LIN {X 0,Y 523.334,Z 556.737,A -85,B 0,C 180,E1 -4767.691,E2 -4767.691} C_VEL
LIN {X 0,Y 523.25,Z 558.343,A -85,B 0,C 180,E1 -4769.23,E2 -4769.23} C_VEL
LIN {X 0,Y 523.25,Z 558.561,A -85,B 0,C 180,E1 -4769.999,E2 -4769.999} C_VEL
LIN {X 0,Y 523.274,Z 557.739,A -85,B 0,C 180,E1 -4771.539,E2 -4771.539} C_VEL
LIN {X 0,Y 523.334,Z 556.746,A -85,B 0,C 180,E1 -4772.308,E2 -4772.308} C_VEL
LIN {X 0,Y 523.367,Z 555.35,A -85,B 0,C 180,E1 -4773.078,E2 -4773.078} C_VEL
LIN {X 0,Y 523.424,Z 552.412,A -85,B 0,C 180,E1 -4774.234,E2 -4774.234} C_VEL
LIN {X 0,Y 523.461,Z 548.433,A -85,B 0,C 180,E1 -4775.392,E2 -4775.392} C_VEL
LIN {X 0,Y 523.514,Z 543.212,A -85,B 0,C 180,E1 -4776.572,E2 -4776.572} C_VEL
LIN {X 0,Y 523.646,Z 536.864,A -85,B 0,C 180,E1 -4777.712,E2 -4777.712} C_VEL
LIN {X 0,Y 523.814,Z 528.822,A -85,B 0,C 180,E1 -4778.875,E2 -4778.875} C_VEL
LIN {X 0,Y 524.043,Z 520.628,A -85,B 0,C 180,E1 -4779.845,E2 -4779.845} C_VEL
LIN {X 0,Y 524.325,Z 510.638,A -85,B 0,C 180,E1 -4780.815,E2 -4780.815} C_VEL
LIN {X 0,Y 524.619,Z 499.337,A -85,B 0,C 180,E1 -4781.691,E2 -4781.691} C_VEL
LIN {X 0,Y 524.85,Z 488.306,A -85,B 0,C 180,E1 -4782.371,E2 -4782.371} C_VEL
LIN {X 0,Y 525.115,Z 476.061,A -85,B 0,C 180,E1 -4782.954,E2 -4782.954} C_VEL
LIN {X 0,Y 525.349,Z 463.204,A -85,B 0,C 180,E1 -4783.391,E2 -4783.391} C_VEL
LIN {X 0,Y 525.549,Z 449.567,A -85,B 0,C 180,E1 -4783.681,E2 -4783.681} C_VEL
LIN {X 0,Y 525.854,Z 356.039,A -85,B 0,C 180,E1 -4784.969,E2 -4784.969} C_VEL
LIN {X 0,Y 524.306,Z 345.568,A -85,B 0,C 180,E1 -4785.178,E2 -4785.178} C_VEL
LIN {X 0,Y 524.738,Z 323.602,A -85,B 0,C 180,E1 -4788.526,E2 -4788.526} C_VEL
LIN {X 0,Y 525.158,Z 305.117,A -85,B 0,C 180,E1 -4791.387,E2 -4791.387} C_VEL
LIN {X 0,Y 525.426,Z 293.296,A -85,B 0,C 180,E1 -4793.239,E2 -4793.239} C_VEL
LIN {X 0,Y 523.993,Z 285.215,A -85,B 0,C 180,E1 -4794.621,E2 -4794.621} C_VEL
LIN {X 0,Y 523.978,Z 285.218,A -85,B 0,C 180,E1 -4797.718,E2 -4797.718} C_VEL
LIN {X 0,Y 523.942,Z 285.215,A -85,B 0,C 180,E1 -4800.854,E2 -4800.854} C_VEL
LIN {X 0,Y 523.958,Z 285.216,A -85,B 0,C 180,E1 -4803.734,E2 -4803.734} C_VEL
LIN {X 0,Y 523.916,Z 285.225,A -85,B 0,C 180,E1 -4806.403,E2 -4806.403} C_VEL
LIN {X 0,Y 523.916,Z 285.218,A -85,B 0,C 180,E1 -4809.084,E2 -4809.084} C_VEL
LIN {X 0,Y 523.95,Z 285.219,A -85,B 0,C 180,E1 -4812.118,E2 -4812.118} C_VEL
LIN {X 0,Y 523.95,Z 285.214,A -85,B 0,C 180,E1 -4815.308,E2 -4815.308} C_VEL
LIN {X 0,Y 523.956,Z 285.221,A -85,B 0,C 180,E1 -4818.688,E2 -4818.688} C_VEL
LIN {X 0,Y 523.912,Z 285.219,A -85,B 0,C 180,E1 -4821.898,E2 -4821.898} C_VEL
LIN {X 0,Y 523.927,Z 285.223,A -85,B 0,C 180,E1 -4824.909,E2 -4824.909} C_VEL
LIN {X 0,Y 523.935,Z 285.215,A -85,B 0,C 180,E1 -4827.678,E2 -4827.678} C_VEL
LIN {X 0,Y 523.955,Z 285.219,A -85,B 0,C 180,E1 -4830.674,E2 -4830.674} C_VEL
LIN {X 0,Y 523.969,Z 285.212,A -85,B 0,C 180,E1 -4833.728,E2 -4833.728} C_VEL
LIN {X 0,Y 523.928,Z 285.217,A -85,B 0,C 180,E1 -4836.27,E2 -4836.27} C_VEL
LIN {X 0,Y 523.937,Z 285.219,A -85,B 0,C 180,E1 -4838.766,E2 -4838.766} C_VEL
LIN {X 0,Y 523.942,Z 285.224,A -85,B 0,C 180,E1 -4841.22,E2 -4841.22} C_VEL
LIN {X 0,Y 523.927,Z 285.22,A -85,B 0,C 180,E1 -4843.639,E2 -4843.639} C_VEL
LIN {X 0,Y 523.936,Z 285.216,A -85,B 0,C 180,E1 -4846.028,E2 -4846.028} C_VEL
LIN {X 0,Y 524.002,Z 285.207,A -85,B 0,C 180,E1 -4848.394,E2 -4848.394} C_VEL
LIN {X 0,Y 523.998,Z 285.217,A -85,B 0,C 180,E1 -4851.516,E2 -4851.516} C_VEL
LIN {X 0,Y 524.074,Z 285.198,A -85,B 0,C 180,E1 -4854.614,E2 -4854.614} C_VEL
LIN {X 0,Y 524.1,Z 285.204,A -85,B 0,C 180,E1 -4857.694,E2 -4857.694} C_VEL
LIN {X 0,Y 524.112,Z 285.193,A -85,B 0,C 180,E1 -4860.768,E2 -4860.768} C_VEL
LIN {X 0,Y 524.064,Z 285.2,A -85,B 0,C 180,E1 -4863.075,E2 -4863.075} C_VEL
LIN {X 0,Y 524.018,Z 285.21,A -85,B 0,C 180,E1 -4866.159,E2 -4866.159} C_VEL
LIN {X 0,Y 523.994,Z 285.21,A -85,B 0,C 180,E1 -4868.484,E2 -4868.484} C_VEL
LIN {X 0,Y 523.992,Z 285.214,A -85,B 0,C 180,E1 -4871.74,E2 -4871.74} C_VEL
LIN {X 0,Y 523.982,Z 285.209,A -85,B 0,C 180,E1 -4875.052,E2 -4875.052} C_VEL
LIN {X 0,Y 523.954,Z 285.22,A -85,B 0,C 180,E1 -4877.969,E2 -4877.969} C_VEL
LIN {X 0,Y 523.962,Z 285.219,A -85,B 0,C 180,E1 -4880.411,E2 -4880.411} C_VEL
LIN {X 0,Y 523.901,Z 285.221,A -85,B 0,C 180,E1 -4882.894,E2 -4882.894} C_VEL
LIN {X 0,Y 523.921,Z 285.217,A -85,B 0,C 180,E1 -4885.421,E2 -4885.421} C_VEL
LIN {X 0,Y 523.944,Z 285.218,A -85,B 0,C 180,E1 -4888.001,E2 -4888.001} C_VEL
LIN {X 0,Y 523.936,Z 285.219,A -85,B 0,C 180,E1 -4890.855,E2 -4890.855} C_VEL
LIN {X 0,Y 523.951,Z 285.214,A -85,B 0,C 180,E1 -4893.735,E2 -4893.735} C_VEL
LIN {X 0,Y 523.895,Z 285.226,A -85,B 0,C 180,E1 -4896.402,E2 -4896.402} C_VEL
LIN {X 0,Y 523.906,Z 285.223,A -85,B 0,C 180,E1 -4899.086,E2 -4899.086} C_VEL
LIN {X 0,Y 523.931,Z 285.217,A -85,B 0,C 180,E1 -4902.121,E2 -4902.121} C_VEL
LIN {X 0,Y 523.934,Z 285.219,A -85,B 0,C 180,E1 -4905.311,E2 -4905.311} C_VEL
LIN {X 0,Y 523.89,Z 285.228,A -85,B 0,C 180,E1 -4906.895,E2 -4906.895} C_VEL
LIN {X 0,Y 523.21,Z 285.308,A -85,B 0,C 180,E1 -4907.536,E2 -4907.536} C_VEL
LIN {X 0,Y 520.359,Z 285.665,A -85,B 0,C 180,E1 -4908.578,E2 -4908.578} C_VEL
LIN {X 0,Y 517.96,Z 285.963,A -85,B 0,C 180,E1 -4909.417,E2 -4909.417} C_VEL
LIN {X 0,Y 516.935,Z 286.088,A -85,B 0,C 180,E1 -4910.065,E2 -4910.065} C_VEL
LIN {X 0,Y 516.853,Z 286.098,A -85,B 0,C 180,E1 -4910.284,E2 -4910.284} C_VEL
LIN {X 0,Y 516.849,Z 286.105,A -85,B 0,C 180,E1 -4913.253,E2 -4913.253} C_VEL
LIN {X 0,Y 516.88,Z 286.094,A -85,B 0,C 180,E1 -4916.12,E2 -4916.12} C_VEL
LIN {X 0,Y 516.877,Z 286.099,A -85,B 0,C 180,E1 -4918.939,E2 -4918.939} C_VEL
LIN {X 0,Y 516.842,Z 286.104,A -85,B 0,C 180,E1 -4921.581,E2 -4921.581} C_VEL
LIN {X 0,Y 516.856,Z 286.097,A -85,B 0,C 180,E1 -4924.208,E2 -4924.208} C_VEL
LIN {X 0,Y 516.855,Z 286.098,A -85,B 0,C 180,E1 -4926.777,E2 -4926.777} C_VEL
LIN {X 0,Y 516.94,Z 286.093,A -85,B 0,C 180,E1 -4929.733,E2 -4929.733} C_VEL
LIN {X 0,Y 516.884,Z 286.094,A -85,B 0,C 180,E1 -4932.595,E2 -4932.595} C_VEL
LIN {X 0,Y 516.933,Z 286.089,A -85,B 0,C 180,E1 -4935.031,E2 -4935.031} C_VEL
LIN {X 0,Y 516.921,Z 286.092,A -85,B 0,C 180,E1 -4938.233,E2 -4938.233} C_VEL
LIN {X 0,Y 516.918,Z 286.095,A -85,B 0,C 180,E1 -4941.4,E2 -4941.4} C_VEL
LIN {X 0,Y 516.984,Z 286.217,A -85,B 0,C 180,E1 -4944.271,E2 -4944.271} C_VEL
LIN {X 0,Y 517.421,Z 290.644,A -85,B 0,C 180,E1 -4945.131,E2 -4945.131} C_VEL
LIN {X 0,Y 517.224,Z 305.053,A -85,B 0,C 180,E1 -4947.859,E2 -4947.859} C_VEL
LIN {X 0,Y 517.167,Z 309.42,A -85,B 0,C 180,E1 -4948.687,E2 -4948.687} C_VEL
LIN {X 0,Y 519.14,Z 320.603,A -85,B 0,C 180,E1 -4948.91,E2 -4948.91} C_VEL
LIN {X 0,Y 518.649,Z 416.692,A -85,B 0,C 180,E1 -4950.267,E2 -4950.267} C_VEL
LIN {X 0,Y 518.394,Z 429.69,A -85,B 0,C 180,E1 -4950.607,E2 -4950.607} C_VEL
LIN {X 0,Y 518.188,Z 442.692,A -85,B 0,C 180,E1 -4951.118,E2 -4951.118} C_VEL
LIN {X 0,Y 517.913,Z 454.471,A -85,B 0,C 180,E1 -4951.75,E2 -4951.75} C_VEL
LIN {X 0,Y 517.589,Z 465.783,A -85,B 0,C 180,E1 -4952.53,E2 -4952.53} C_VEL
LIN {X 0,Y 517.331,Z 475.987,A -85,B 0,C 180,E1 -4953.408,E2 -4953.408} C_VEL
LIN {X 0,Y 517.031,Z 484.379,A -85,B 0,C 180,E1 -4954.288,E2 -4954.288} C_VEL
LIN {X 0,Y 516.788,Z 493.475,A -85,B 0,C 180,E1 -4955.463,E2 -4955.463} C_VEL
LIN {X 0,Y 516.584,Z 501.205,A -85,B 0,C 180,E1 -4956.709,E2 -4956.709} C_VEL
LIN {X 0,Y 516.46,Z 506.722,A -85,B 0,C 180,E1 -4957.822,E2 -4957.822} C_VEL
LIN {X 0,Y 516.359,Z 511.397,A -85,B 0,C 180,E1 -4959.006,E2 -4959.006} C_VEL
LIN {X 0,Y 516.319,Z 514.967,A -85,B 0,C 180,E1 -4960.193,E2 -4960.193} C_VEL
LIN {X 0,Y 516.287,Z 517.639,A -85,B 0,C 180,E1 -4961.447,E2 -4961.447} C_VEL
LIN {X 0,Y 516.182,Z 519.129,A -85,B 0,C 180,E1 -4962.583,E2 -4962.583} C_VEL
LIN {X 0,Y 516.178,Z 519.7,A -85,B 0,C 180,E1 -4963.384,E2 -4963.384} C_VEL
LIN {X 0,Y 516.206,Z 519.621,A -85,B 0,C 180,E1 -4964.839,E2 -4964.839} C_VEL
LIN {X 0,Y 516.143,Z 518.833,A -85,B 0,C 180,E1 -4965.803,E2 -4965.803} C_VEL
LIN {X 0,Y 516.189,Z 517.703,A -85,B 0,C 180,E1 -4966.614,E2 -4966.614} C_VEL
LIN {X 0,Y 516.277,Z 515.579,A -85,B 0,C 180,E1 -4967.654,E2 -4967.654} C_VEL
LIN {X 0,Y 516.357,Z 511.48,A -85,B 0,C 180,E1 -4969.066,E2 -4969.066} C_VEL
LIN {X 0,Y 516.511,Z 506.399,A -85,B 0,C 180,E1 -4970.343,E2 -4970.343} C_VEL
LIN {X 0,Y 516.581,Z 500.268,A -85,B 0,C 180,E1 -4971.551,E2 -4971.551} C_VEL
LIN {X 0,Y 516.861,Z 492.303,A -85,B 0,C 180,E1 -4972.801,E2 -4972.801} C_VEL
LIN {X 0,Y 517.045,Z 483.958,A -85,B 0,C 180,E1 -4973.853,E2 -4973.853} C_VEL
LIN {X 0,Y 517.331,Z 473.616,A -85,B 0,C 180,E1 -4974.907,E2 -4974.907} C_VEL
LIN {X 0,Y 517.645,Z 463.336,A -85,B 0,C 180,E1 -4975.751,E2 -4975.751} C_VEL
LIN {X 0,Y 518.018,Z 451.513,A -85,B 0,C 180,E1 -4976.516,E2 -4976.516} C_VEL
LIN {X 0,Y 518.229,Z 439.172,A -85,B 0,C 180,E1 -4977.13,E2 -4977.13} C_VEL
LIN {X 0,Y 518.434,Z 426.616,A -85,B 0,C 180,E1 -4977.583,E2 -4977.583} C_VEL
LIN {X 0,Y 518.598,Z 413.993,A -85,B 0,C 180,E1 -4977.875,E2 -4977.875} C_VEL
LIN {X 0,Y 519.041,Z 319.422,A -85,B 0,C 180,E1 -4979.201,E2 -4979.201} C_VEL
LIN {X 0,Y 517.209,Z 309.191,A -85,B 0,C 180,E1 -4979.426,E2 -4979.426} C_VEL
LIN {X 0,Y 517.372,Z 293.368,A -85,B 0,C 180,E1 -4982.31,E2 -4982.31} C_VEL
LIN {X 0,Y 517.178,Z 287.47,A -85,B 0,C 180,E1 -4983.392,E2 -4983.392} C_VEL
LIN {X 0,Y 516.938,Z 286.096,A -85,B 0,C 180,E1 -4983.672,E2 -4983.672} C_VEL
LIN {X 0,Y 516.879,Z 286.098,A -85,B 0,C 180,E1 -4986.746,E2 -4986.746} C_VEL
LIN {X 0,Y 516.884,Z 286.096,A -85,B 0,C 180,E1 -4989.721,E2 -4989.721} C_VEL
LIN {X 0,Y 516.914,Z 286.093,A -85,B 0,C 180,E1 -4991.775,E2 -4991.775} C_VEL
LIN {X 0,Y 516.897,Z 286.097,A -85,B 0,C 180,E1 -4995.007,E2 -4995.007} C_VEL
LIN {X 0,Y 516.915,Z 286.098,A -85,B 0,C 180,E1 -4998.399,E2 -4998.399} C_VEL
LIN {X 0,Y 516.881,Z 286.096,A -85,B 0,C 180,E1 -5001.284,E2 -5001.284} C_VEL
LIN {X 0,Y 516.872,Z 286.098,A -85,B 0,C 180,E1 -5004.219,E2 -5004.219} C_VEL
LIN {X 0,Y 516.895,Z 286.1,A -85,B 0,C 180,E1 -5007.053,E2 -5007.053} C_VEL
LIN {X 0,Y 516.892,Z 286.092,A -85,B 0,C 180,E1 -5009.796,E2 -5009.796} C_VEL
LIN {X 0,Y 516.926,Z 286.09,A -85,B 0,C 180,E1 -5012.467,E2 -5012.467} C_VEL
LIN {X 0,Y 516.909,Z 286.099,A -85,B 0,C 180,E1 -5015.072,E2 -5015.072} C_VEL
LIN {X 0,Y 516.885,Z 286.094,A -85,B 0,C 180,E1 -5018.462,E2 -5018.462} C_VEL
LIN {X 0,Y 516.901,Z 286.094,A -85,B 0,C 180,E1 -5020.955,E2 -5020.955} C_VEL
LIN {X 0,Y 516.914,Z 286.099,A -85,B 0,C 180,E1 -5023.41,E2 -5023.41} C_VEL
LIN {X 0,Y 516.894,Z 286.096,A -85,B 0,C 180,E1 -5025.834,E2 -5025.834} C_VEL
LIN {X 0,Y 516.966,Z 286.085,A -85,B 0,C 180,E1 -5028.234,E2 -5028.234} C_VEL
LIN {X 0,Y 516.967,Z 286.085,A -85,B 0,C 180,E1 -5031.4,E2 -5031.4} C_VEL
LIN {X 0,Y 517.002,Z 286.088,A -85,B 0,C 180,E1 -5033.757,E2 -5033.757} C_VEL
LIN {X 0,Y 517.012,Z 286.076,A -85,B 0,C 180,E1 -5036.883,E2 -5036.883} C_VEL
LIN {X 0,Y 517.085,Z 286.074,A -85,B 0,C 180,E1 -5040,E2 -5040} C_VEL
LIN {X 0,Y 517.012,Z 286.077,A -85,B 0,C 180,E1 -5043.117,E2 -5043.117} C_VEL
LIN {X 0,Y 517.002,Z 286.084,A -85,B 0,C 180,E1 -5046.243,E2 -5046.243} C_VEL
LIN {X 0,Y 516.945,Z 286.086,A -85,B 0,C 180,E1 -5049.389,E2 -5049.389} C_VEL
LIN {X 0,Y 516.951,Z 286.083,A -85,B 0,C 180,E1 -5051.807,E2 -5051.807} C_VEL
LIN {X 0,Y 516.944,Z 286.085,A -85,B 0,C 180,E1 -5055.146,E2 -5055.146} C_VEL
LIN {X 0,Y 516.924,Z 286.093,A -85,B 0,C 180,E1 -5058.222,E2 -5058.222} C_VEL
LIN {X 0,Y 516.912,Z 286.096,A -85,B 0,C 180,E1 -5060.702,E2 -5060.702} C_VEL
LIN {X 0,Y 516.903,Z 286.093,A -85,B 0,C 180,E1 -5064.072,E2 -5064.072} C_VEL
LIN {X 0,Y 516.924,Z 286.093,A -85,B 0,C 180,E1 -5066.658,E2 -5066.658} C_VEL
LIN {X 0,Y 516.911,Z 286.089,A -85,B 0,C 180,E1 -5069.524,E2 -5069.524} C_VEL
LIN {X 0,Y 516.894,Z 286.096,A -85,B 0,C 180,E1 -5072.543,E2 -5072.543} C_VEL
LIN {X 0,Y 516.865,Z 286.102,A -85,B 0,C 180,E1 -5075.33,E2 -5075.33} C_VEL
LIN {X 0,Y 516.881,Z 286.095,A -85,B 0,C 180,E1 -5077.943,E2 -5077.943} C_VEL
LIN {X 0,Y 516.884,Z 286.096,A -85,B 0,C 180,E1 -5080.742,E2 -5080.742} C_VEL
LIN {X 0,Y 516.883,Z 286.097,A -85,B 0,C 180,E1 -5082.832,E2 -5082.832} C_VEL
LIN {X 0,Y 516.896,Z 286.097,A -85,B 0,C 180,E1 -5085.007,E2 -5085.007} C_VEL
LIN {X 0,Y 516.915,Z 286.091,A -85,B 0,C 180,E1 -5088.399,E2 -5088.399} C_VEL
LIN {X 0,Y 516.882,Z 286.097,A -85,B 0,C 180,E1 -5091.284,E2 -5091.284} C_VEL
LIN {X 0,Y 516.873,Z 286.098,A -85,B 0,C 180,E1 -5094.22,E2 -5094.22} C_VEL
LIN {X 0,Y 516.897,Z 286.092,A -85,B 0,C 180,E1 -5097.053,E2 -5097.053} C_VEL
LIN {X 0,Y 516.895,Z 286.101,A -85,B 0,C 180,E1 -5099.796,E2 -5099.796} C_VEL
LIN {X 0,Y 516.927,Z 286.095,A -85,B 0,C 180,E1 -5102.467,E2 -5102.467} C_VEL
LIN {X 0,Y 516.968,Z 286.253,A -85,B 0,C 180,E1 -5105.337,E2 -5105.337} C_VEL
LIN {X 0,Y 518.473,Z 295.27,A -85,B 0,C 180,E1 -5106.852,E2 -5106.852} C_VEL
LIN {X 0,Y 517.947,Z 315.172,A -85,B 0,C 180,E1 -5109.977,E2 -5109.977} C_VEL
LIN {X 0,Y 517.471,Z 333.541,A -85,B 0,C 180,E1 -5112.818,E2 -5112.818} C_VEL
LIN {X 0,Y 517.285,Z 345.531,A -85,B 0,C 180,E1 -5114.635,E2 -5114.635} C_VEL
LIN {X 0,Y 519.028,Z 357.668,A -85,B 0,C 180,E1 -5114.857,E2 -5114.857} C_VEL
LIN {X 0,Y 518.61,Z 453.531,A -85,B 0,C 180,E1 -5116.206,E2 -5116.206} C_VEL
LIN {X 0,Y 518.365,Z 466.892,A -85,B 0,C 180,E1 -5116.549,E2 -5116.549} C_VEL
LIN {X 0,Y 518.053,Z 480.235,A -85,B 0,C 180,E1 -5117.065,E2 -5117.065} C_VEL
LIN {X 0,Y 517.807,Z 492.308,A -85,B 0,C 180,E1 -5117.711,E2 -5117.711} C_VEL
LIN {X 0,Y 517.514,Z 504.366,A -85,B 0,C 180,E1 -5118.544,E2 -5118.544} C_VEL
LIN {X 0,Y 517.17,Z 514.592,A -85,B 0,C 180,E1 -5119.428,E2 -5119.428} C_VEL
LIN {X 0,Y 516.891,Z 523.792,A -85,B 0,C 180,E1 -5120.412,E2 -5120.412} C_VEL
LIN {X 0,Y 516.658,Z 532.759,A -85,B 0,C 180,E1 -5121.591,E2 -5121.591} C_VEL
LIN {X 0,Y 516.505,Z 539.977,A -85,B 0,C 180,E1 -5122.769,E2 -5122.769} C_VEL
LIN {X 0,Y 516.419,Z 546.553,A -85,B 0,C 180,E1 -5124.141,E2 -5124.141} C_VEL
LIN {X 0,Y 516.269,Z 550.9,A -85,B 0,C 180,E1 -5125.314,E2 -5125.314} C_VEL
LIN {X 0,Y 516.352,Z 553.207,A -85,B 0,C 180,E1 -5126.097,E2 -5126.097} C_VEL
LIN {X 0,Y 516.282,Z 555.072,A -85,B 0,C 180,E1 -5126.878,E2 -5126.878} C_VEL
LIN {X 0,Y 516.26,Z 556.472,A -85,B 0,C 180,E1 -5127.659,E2 -5127.659} C_VEL
LIN {X 0,Y 516.16,Z 558.079,A -85,B 0,C 180,E1 -5129.219,E2 -5129.219} C_VEL
LIN {X 0,Y 516.158,Z 558.297,A -85,B 0,C 180,E1 -5129.999,E2 -5129.999} C_VEL
LIN {X 0,Y 516.191,Z 557.476,A -85,B 0,C 180,E1 -5131.56,E2 -5131.56} C_VEL
LIN {X 0,Y 516.26,Z 556.483,A -85,B 0,C 180,E1 -5132.34,E2 -5132.34} C_VEL
LIN {X 0,Y 516.282,Z 555.086,A -85,B 0,C 180,E1 -5133.121,E2 -5133.121} C_VEL
LIN {X 0,Y 516.312,Z 552.147,A -85,B 0,C 180,E1 -5134.293,E2 -5134.293} C_VEL
LIN {X 0,Y 516.375,Z 548.168,A -85,B 0,C 180,E1 -5135.466,E2 -5135.466} C_VEL
LIN {X 0,Y 516.45,Z 542.252,A -85,B 0,C 180,E1 -5136.798,E2 -5136.798} C_VEL
LIN {X 0,Y 516.596,Z 535.358,A -85,B 0,C 180,E1 -5138.015,E2 -5138.015} C_VEL
LIN {X 0,Y 516.811,Z 527.06,A -85,B 0,C 180,E1 -5139.194,E2 -5139.194} C_VEL
LIN {X 0,Y 517.039,Z 518.555,A -85,B 0,C 180,E1 -5140.177,E2 -5140.177} C_VEL
LIN {X 0,Y 517.369,Z 508.047,A -85,B 0,C 180,E1 -5141.161,E2 -5141.161} C_VEL
LIN {X 0,Y 517.71,Z 496.582,A -85,B 0,C 180,E1 -5142.022,E2 -5142.022} C_VEL
LIN {X 0,Y 517.941,Z 486.258,A -85,B 0,C 180,E1 -5142.638,E2 -5142.638} C_VEL
LIN {X 0,Y 518.21,Z 474.559,A -85,B 0,C 180,E1 -5143.179,E2 -5143.179} C_VEL
LIN {X 0,Y 518.468,Z 461.083,A -85,B 0,C 180,E1 -5143.622,E2 -5143.622} C_VEL
LIN {X 0,Y 518.681,Z 447.723,A -85,B 0,C 180,E1 -5143.891,E2 -5143.891} C_VEL
LIN {X 0,Y 518.913,Z 356.099,A -85,B 0,C 180,E1 -5145.169,E2 -5145.169} C_VEL
LIN {X 0,Y 517.274,Z 345.383,A -85,B 0,C 180,E1 -5145.377,E2 -5145.377} C_VEL
LIN {X 0,Y 517.746,Z 324.527,A -85,B 0,C 180,E1 -5148.601,E2 -5148.601} C_VEL
LIN {X 0,Y 518.196,Z 306.176,A -85,B 0,C 180,E1 -5151.48,E2 -5151.48} C_VEL
LIN {X 0,Y 518.458,Z 294.337,A -85,B 0,C 180,E1 -5153.359,E2 -5153.359} C_VEL
LIN {X 0,Y 516.939,Z 286.094,A -85,B 0,C 180,E1 -5154.781,E2 -5154.781} C_VEL
LIN {X 0,Y 516.926,Z 286.098,A -85,B 0,C 180,E1 -5157.905,E2 -5157.905} C_VEL
LIN {X 0,Y 516.89,Z 286.103,A -85,B 0,C 180,E1 -5160.203,E2 -5160.203} C_VEL
LIN {X 0,Y 516.892,Z 286.093,A -85,B 0,C 180,E1 -5162.946,E2 -5162.946} C_VEL
LIN {X 0,Y 516.884,Z 286.097,A -85,B 0,C 180,E1 -5165.778,E2 -5165.778} C_VEL
LIN {X 0,Y 516.877,Z 286.098,A -85,B 0,C 180,E1 -5168.715,E2 -5168.715} C_VEL
LIN {X 0,Y 516.909,Z 286.092,A -85,B 0,C 180,E1 -5171.774,E2 -5171.774} C_VEL
LIN {X 0,Y 516.917,Z 286.092,A -85,B 0,C 180,E1 -5175.009,E2 -5175.009} C_VEL
LIN {X 0,Y 516.911,Z 286.097,A -85,B 0,C 180,E1 -5178.397,E2 -5178.397} C_VEL
LIN {X 0,Y 516.877,Z 286.096,A -85,B 0,C 180,E1 -5181.284,E2 -5181.284} C_VEL
LIN {X 0,Y 516.88,Z 286.097,A -85,B 0,C 180,E1 -5184.22,E2 -5184.22} C_VEL
LIN {X 0,Y 516.89,Z 286.099,A -85,B 0,C 180,E1 -5187.053,E2 -5187.053} C_VEL
LIN {X 0,Y 516.893,Z 286.093,A -85,B 0,C 180,E1 -5189.796,E2 -5189.796} C_VEL
LIN {X 0,Y 516.921,Z 286.092,A -85,B 0,C 180,E1 -5192.467,E2 -5192.467} C_VEL
LIN {X 0,Y 516.903,Z 286.1,A -85,B 0,C 180,E1 -5195.071,E2 -5195.071} C_VEL
LIN {X 0,Y 516.877,Z 286.096,A -85,B 0,C 180,E1 -5198.462,E2 -5198.462} C_VEL
LIN {X 0,Y 516.894,Z 286.099,A -85,B 0,C 180,E1 -5200.954,E2 -5200.954} C_VEL
LIN {X 0,Y 516.904,Z 286.098,A -85,B 0,C 180,E1 -5203.41,E2 -5203.41} C_VEL
LIN {X 0,Y 516.897,Z 286.094,A -85,B 0,C 180,E1 -5205.834,E2 -5205.834} C_VEL
LIN {X 0,Y 516.947,Z 286.09,A -85,B 0,C 180,E1 -5209.028,E2 -5209.028} C_VEL
LIN {X 0,Y 516.969,Z 286.084,A -85,B 0,C 180,E1 -5212.187,E2 -5212.187} C_VEL
LIN {X 0,Y 517.021,Z 286.077,A -85,B 0,C 180,E1 -5214.54,E2 -5214.54} C_VEL
LIN {X 0,Y 517.072,Z 286.08,A -85,B 0,C 180,E1 -5217.663,E2 -5217.663} C_VEL
LIN {X 0,Y 517.083,Z 286.069,A -85,B 0,C 180,E1 -5220.779,E2 -5220.779} C_VEL
LIN {X 0,Y 517.005,Z 286.08,A -85,B 0,C 180,E1 -5223.117,E2 -5223.117} C_VEL
LIN {X 0,Y 516.98,Z 286.085,A -85,B 0,C 180,E1 -5226.244,E2 -5226.244} C_VEL
LIN {X 0,Y 516.958,Z 286.085,A -85,B 0,C 180,E1 -5228.601,E2 -5228.601} C_VEL
LIN {X 0,Y 516.942,Z 286.093,A -85,B 0,C 180,E1 -5231.807,E2 -5231.807} C_VEL
LIN {X 0,Y 516.933,Z 286.088,A -85,B 0,C 180,E1 -5235.146,E2 -5235.146} C_VEL
LIN {X 0,Y 516.915,Z 286.099,A -85,B 0,C 180,E1 -5238.223,E2 -5238.223} C_VEL
LIN {X 0,Y 516.902,Z 286.094,A -85,B 0,C 180,E1 -5240.702,E2 -5240.702} C_VEL
LIN {X 0,Y 516.881,Z 286.1,A -85,B 0,C 180,E1 -5244.074,E2 -5244.074} C_VEL
LIN {X 0,Y 516.895,Z 286.098,A -85,B 0,C 180,E1 -5246.66,E2 -5246.66} C_VEL
LIN {X 0,Y 516.902,Z 286.091,A -85,B 0,C 180,E1 -5249.524,E2 -5249.524} C_VEL
LIN {X 0,Y 516.887,Z 286.103,A -85,B 0,C 180,E1 -5252.544,E2 -5252.544} C_VEL
LIN {X 0,Y 516.858,Z 286.098,A -85,B 0,C 180,E1 -5255.33,E2 -5255.33} C_VEL
LIN {X 0,Y 516.872,Z 286.096,A -85,B 0,C 180,E1 -5257.944,E2 -5257.944} C_VEL
LIN {X 0,Y 516.857,Z 286.107,A -85,B 0,C 180,E1 -5260.744,E2 -5260.744} C_VEL
LIN {X 0,Y 516.848,Z 286.108,A -85,B 0,C 180,E1 -5262.835,E2 -5262.835} C_VEL
LIN {X 0,Y 516.89,Z 286.101,A -85,B 0,C 180,E1 -5265.008,E2 -5265.008} C_VEL
LIN {X 0,Y 516.883,Z 286.096,A -85,B 0,C 180,E1 -5268.403,E2 -5268.403} C_VEL
LIN {X 0,Y 516.853,Z 286.098,A -85,B 0,C 180,E1 -5270.284,E2 -5270.284} C_VEL
LIN {X 0,Y 516.192,Z 286.188,A -85,B 0,C 180,E1 -5270.934,E2 -5270.934} C_VEL
LIN {X 0,Y 513.345,Z 286.542,A -85,B 0,C 180,E1 -5271.99,E2 -5271.99} C_VEL
LIN {X 0,Y 510.932,Z 286.842,A -85,B 0,C 180,E1 -5272.84,E2 -5272.84} C_VEL
LIN {X 0,Y 509.89,Z 286.969,A -85,B 0,C 180,E1 -5273.497,E2 -5273.497} C_VEL
LIN {X 0,Y 509.802,Z 286.977,A -85,B 0,C 180,E1 -5273.719,E2 -5273.719} C_VEL
LIN {X 0,Y 509.838,Z 286.973,A -85,B 0,C 180,E1 -5276.539,E2 -5276.539} C_VEL
LIN {X 0,Y 509.825,Z 286.982,A -85,B 0,C 180,E1 -5279.334,E2 -5279.334} C_VEL
LIN {X 0,Y 509.825,Z 286.974,A -85,B 0,C 180,E1 -5282.052,E2 -5282.052} C_VEL
LIN {X 0,Y 509.793,Z 286.978,A -85,B 0,C 180,E1 -5284.701,E2 -5284.701} C_VEL
LIN {X 0,Y 509.825,Z 286.983,A -85,B 0,C 180,E1 -5287.459,E2 -5287.459} C_VEL
LIN {X 0,Y 509.916,Z 286.966,A -85,B 0,C 180,E1 -5289.846,E2 -5289.846} C_VEL
LIN {X 0,Y 509.851,Z 286.973,A -85,B 0,C 180,E1 -5293.174,E2 -5293.174} C_VEL
LIN {X 0,Y 509.847,Z 286.979,A -85,B 0,C 180,E1 -5295.634,E2 -5295.634} C_VEL
LIN {X 0,Y 509.856,Z 286.969,A -85,B 0,C 180,E1 -5298.874,E2 -5298.874} C_VEL
LIN {X 0,Y 509.875,Z 286.977,A -85,B 0,C 180,E1 -5302.078,E2 -5302.078} C_VEL
LIN {X 0,Y 509.965,Z 287.173,A -85,B 0,C 180,E1 -5304.167,E2 -5304.167} C_VEL
LIN {X 0,Y 510.428,Z 291.743,A -85,B 0,C 180,E1 -5305.064,E2 -5305.064} C_VEL
LIN {X 0,Y 510.252,Z 305.212,A -85,B 0,C 180,E1 -5307.632,E2 -5307.632} C_VEL
LIN {X 0,Y 510.172,Z 309.624,A -85,B 0,C 180,E1 -5308.471,E2 -5308.471} C_VEL
LIN {X 0,Y 512.24,Z 320.694,A -85,B 0,C 180,E1 -5308.698,E2 -5308.698} C_VEL
LIN {X 0,Y 511.789,Z 416.698,A -85,B 0,C 180,E1 -5310.074,E2 -5310.074} C_VEL
LIN {X 0,Y 511.544,Z 429.022,A -85,B 0,C 180,E1 -5310.394,E2 -5310.394} C_VEL
LIN {X 0,Y 511.292,Z 441.742,A -85,B 0,C 180,E1 -5310.887,E2 -5310.887} C_VEL
LIN {X 0,Y 511.038,Z 453.052,A -85,B 0,C 180,E1 -5311.478,E2 -5311.478} C_VEL
LIN {X 0,Y 510.672,Z 464.708,A -85,B 0,C 180,E1 -5312.268,E2 -5312.268} C_VEL
LIN {X 0,Y 510.334,Z 475.156,A -85,B 0,C 180,E1 -5313.158,E2 -5313.158} C_VEL
LIN {X 0,Y 510.017,Z 484.603,A -85,B 0,C 180,E1 -5314.149,E2 -5314.149} C_VEL
LIN {X 0,Y 509.745,Z 493.71,A -85,B 0,C 180,E1 -5315.34,E2 -5315.34} C_VEL
LIN {X 0,Y 509.578,Z 500.854,A -85,B 0,C 180,E1 -5316.499,E2 -5316.499} C_VEL
LIN {X 0,Y 509.431,Z 506.058,A -85,B 0,C 180,E1 -5317.531,E2 -5317.531} C_VEL
LIN {X 0,Y 509.316,Z 510.927,A -85,B 0,C 180,E1 -5318.731,E2 -5318.731} C_VEL
LIN {X 0,Y 509.256,Z 514.68,A -85,B 0,C 180,E1 -5319.934,E2 -5319.934} C_VEL
LIN {X 0,Y 509.191,Z 518.039,A -85,B 0,C 180,E1 -5321.488,E2 -5321.488} C_VEL
LIN {X 0,Y 509.103,Z 519.587,A -85,B 0,C 180,E1 -5322.761,E2 -5322.761} C_VEL
LIN {X 0,Y 509.085,Z 520.017,A -85,B 0,C 180,E1 -5323.574,E2 -5323.574} C_VEL
LIN {X 0,Y 509.121,Z 519.845,A -85,B 0,C 180,E1 -5324.917,E2 -5324.917} C_VEL
LIN {X 0,Y 509.055,Z 518.868,A -85,B 0,C 180,E1 -5326.029,E2 -5326.029} C_VEL
LIN {X 0,Y 509.116,Z 517.6,A -85,B 0,C 180,E1 -5326.852,E2 -5326.852} C_VEL
LIN {X 0,Y 509.204,Z 515.719,A -85,B 0,C 180,E1 -5327.761,E2 -5327.761} C_VEL
LIN {X 0,Y 509.274,Z 512.444,A -85,B 0,C 180,E1 -5328.924,E2 -5328.924} C_VEL
LIN {X 0,Y 509.427,Z 507.43,A -85,B 0,C 180,E1 -5330.261,E2 -5330.261} C_VEL
LIN {X 0,Y 509.551,Z 500.555,A -85,B 0,C 180,E1 -5331.651,E2 -5331.651} C_VEL
LIN {X 0,Y 509.836,Z 492.593,A -85,B 0,C 180,E1 -5332.919,E2 -5332.919} C_VEL
LIN {X 0,Y 510.06,Z 484.258,A -85,B 0,C 180,E1 -5333.984,E2 -5333.984} C_VEL
LIN {X 0,Y 510.336,Z 475.562,A -85,B 0,C 180,E1 -5334.898,E2 -5334.898} C_VEL
LIN {X 0,Y 510.675,Z 465.037,A -85,B 0,C 180,E1 -5335.8,E2 -5335.8} C_VEL
LIN {X 0,Y 511.05,Z 454.324,A -85,B 0,C 180,E1 -5336.536,E2 -5336.536} C_VEL
LIN {X 0,Y 511.283,Z 441.958,A -85,B 0,C 180,E1 -5337.197,E2 -5337.197} C_VEL
LIN {X 0,Y 511.55,Z 428.714,A -85,B 0,C 180,E1 -5337.708,E2 -5337.708} C_VEL
LIN {X 0,Y 511.713,Z 416.293,A -85,B 0,C 180,E1 -5338.028,E2 -5338.028} C_VEL
LIN {X 0,Y 512.221,Z 320.593,A -85,B 0,C 180,E1 -5339.395,E2 -5339.395} C_VEL
LIN {X 0,Y 510.216,Z 309.524,A -85,B 0,C 180,E1 -5339.617,E2 -5339.617} C_VEL
LIN {X 0,Y 510.408,Z 292.85,A -85,B 0,C 180,E1 -5342.675,E2 -5342.675} C_VEL
LIN {X 0,Y 509.899,Z 286.973,A -85,B 0,C 180,E1 -5343.784,E2 -5343.784} C_VEL
LIN {X 0,Y 509.821,Z 286.976,A -85,B 0,C 180,E1 -5346.913,E2 -5346.913} C_VEL
LIN {X 0,Y 509.836,Z 286.974,A -85,B 0,C 180,E1 -5349.47,E2 -5349.47} C_VEL
LIN {X 0,Y 509.835,Z 286.981,A -85,B 0,C 180,E1 -5352.49,E2 -5352.49} C_VEL
LIN {X 0,Y 509.841,Z 286.974,A -85,B 0,C 180,E1 -5355.33,E2 -5355.33} C_VEL
LIN {X 0,Y 509.857,Z 286.98,A -85,B 0,C 180,E1 -5358.574,E2 -5358.574} C_VEL
LIN {X 0,Y 509.852,Z 286.97,A -85,B 0,C 180,E1 -5361.786,E2 -5361.786} C_VEL
LIN {X 0,Y 509.831,Z 286.98,A -85,B 0,C 180,E1 -5364.622,E2 -5364.622} C_VEL
LIN {X 0,Y 509.862,Z 286.971,A -85,B 0,C 180,E1 -5367.481,E2 -5367.481} C_VEL
LIN {X 0,Y 509.859,Z 286.968,A -85,B 0,C 180,E1 -5370.274,E2 -5370.274} C_VEL
LIN {X 0,Y 509.884,Z 286.974,A -85,B 0,C 180,E1 -5372.944,E2 -5372.944} C_VEL
LIN {X 0,Y 509.865,Z 286.972,A -85,B 0,C 180,E1 -5375.574,E2 -5375.574} C_VEL
LIN {X 0,Y 509.85,Z 286.975,A -85,B 0,C 180,E1 -5378.998,E2 -5378.998} C_VEL
LIN {X 0,Y 509.882,Z 286.967,A -85,B 0,C 180,E1 -5382.001,E2 -5382.001} C_VEL
LIN {X 0,Y 509.911,Z 286.963,A -85,B 0,C 180,E1 -5384.819,E2 -5384.819} C_VEL
LIN {X 0,Y 509.9,Z 286.966,A -85,B 0,C 180,E1 -5388.124,E2 -5388.124} C_VEL
LIN {X 0,Y 509.914,Z 286.962,A -85,B 0,C 180,E1 -5391.28,E2 -5391.28} C_VEL
LIN {X 0,Y 509.953,Z 286.966,A -85,B 0,C 180,E1 -5393.67,E2 -5393.67} C_VEL
LIN {X 0,Y 510.054,Z 286.949,A -85,B 0,C 180,E1 -5397.631,E2 -5397.631} C_VEL
LIN {X 0,Y 510.062,Z 286.939,A -85,B 0,C 180,E1 -5400.789,E2 -5400.789} C_VEL
LIN {X 0,Y 509.954,Z 286.957,A -85,B 0,C 180,E1 -5403.16,E2 -5403.16} C_VEL
LIN {X 0,Y 509.953,Z 286.962,A -85,B 0,C 180,E1 -5406.33,E2 -5406.33} C_VEL
LIN {X 0,Y 509.911,Z 286.965,A -85,B 0,C 180,E1 -5408.72,E2 -5408.72} C_VEL
LIN {X 0,Y 509.904,Z 286.962,A -85,B 0,C 180,E1 -5411.932,E2 -5411.932} C_VEL
LIN {X 0,Y 509.894,Z 286.963,A -85,B 0,C 180,E1 -5415.242,E2 -5415.242} C_VEL
LIN {X 0,Y 509.882,Z 286.967,A -85,B 0,C 180,E1 -5417.998,E2 -5417.998} C_VEL
LIN {X 0,Y 509.85,Z 286.972,A -85,B 0,C 180,E1 -5421.002,E2 -5421.002} C_VEL
LIN {X 0,Y 509.864,Z 286.974,A -85,B 0,C 180,E1 -5424.426,E2 -5424.426} C_VEL
LIN {X 0,Y 509.884,Z 286.972,A -85,B 0,C 180,E1 -5427.056,E2 -5427.056} C_VEL
LIN {X 0,Y 509.858,Z 286.966,A -85,B 0,C 180,E1 -5429.751,E2 -5429.751} C_VEL
LIN {X 0,Y 509.867,Z 286.974,A -85,B 0,C 180,E1 -5432.773,E2 -5432.773} C_VEL
LIN {X 0,Y 509.825,Z 286.976,A -85,B 0,C 180,E1 -5435.578,E2 -5435.578} C_VEL
LIN {X 0,Y 509.85,Z 286.97,A -85,B 0,C 180,E1 -5438.338,E2 -5438.338} C_VEL
LIN {X 0,Y 509.856,Z 286.978,A -85,B 0,C 180,E1 -5441.426,E2 -5441.426} C_VEL
LIN {X 0,Y 509.84,Z 286.973,A -85,B 0,C 180,E1 -5444.67,E2 -5444.67} C_VEL
LIN {X 0,Y 509.857,Z 286.972,A -85,B 0,C 180,E1 -5448.103,E2 -5448.103} C_VEL
LIN {X 0,Y 509.847,Z 286.969,A -85,B 0,C 180,E1 -5450.648,E2 -5450.648} C_VEL
LIN {X 0,Y 509.827,Z 286.98,A -85,B 0,C 180,E1 -5453.647,E2 -5453.647} C_VEL
LIN {X 0,Y 509.861,Z 286.969,A -85,B 0,C 180,E1 -5456.539,E2 -5456.539} C_VEL
LIN {X 0,Y 509.848,Z 286.973,A -85,B 0,C 180,E1 -5459.334,E2 -5459.334} C_VEL
LIN {X 0,Y 509.892,Z 286.973,A -85,B 0,C 180,E1 -5462.054,E2 -5462.054} C_VEL
LIN {X 0,Y 509.918,Z 286.989,A -85,B 0,C 180,E1 -5465.131,E2 -5465.131} C_VEL
LIN {X 0,Y 511.538,Z 296.955,A -85,B 0,C 180,E1 -5466.833,E2 -5466.833} C_VEL
LIN {X 0,Y 510.957,Z 316.127,A -85,B 0,C 180,E1 -5469.887,E2 -5469.887} C_VEL
LIN {X 0,Y 510.462,Z 334.573,A -85,B 0,C 180,E1 -5472.782,E2 -5472.782} C_VEL
LIN {X 0,Y 510.265,Z 345.203,A -85,B 0,C 180,E1 -5474.417,E2 -5474.417} C_VEL
LIN {X 0,Y 512.162,Z 358.326,A -85,B 0,C 180,E1 -5474.662,E2 -5474.662} C_VEL
LIN {X 0,Y 511.72,Z 453.215,A -85,B 0,C 180,E1 -5476.017,E2 -5476.017} C_VEL
LIN {X 0,Y 511.446,Z 466.591,A -85,B 0,C 180,E1 -5476.364,E2 -5476.364} C_VEL
LIN {X 0,Y 511.14,Z 479.943,A -85,B 0,C 180,E1 -5476.887,E2 -5476.887} C_VEL
LIN {X 0,Y 510.846,Z 491.402,A -85,B 0,C 180,E1 -5477.502,E2 -5477.502} C_VEL
LIN {X 0,Y 510.554,Z 502.785,A -85,B 0,C 180,E1 -5478.285,E2 -5478.285} C_VEL
LIN {X 0,Y 510.222,Z 513.262,A -85,B 0,C 180,E1 -5479.182,E2 -5479.182} C_VEL
LIN {X 0,Y 509.923,Z 521.829,A -85,B 0,C 180,E1 -5480.079,E2 -5480.079} C_VEL
LIN {X 0,Y 509.666,Z 529.735,A -85,B 0,C 180,E1 -5481.075,E2 -5481.075} C_VEL
LIN {X 0,Y 509.48,Z 537.459,A -85,B 0,C 180,E1 -5482.27,E2 -5482.27} C_VEL
LIN {X 0,Y 509.308,Z 544.578,A -85,B 0,C 180,E1 -5483.662,E2 -5483.662} C_VEL
LIN {X 0,Y 509.243,Z 549.316,A -85,B 0,C 180,E1 -5484.853,E2 -5484.853} C_VEL
LIN {X 0,Y 509.246,Z 552.938,A -85,B 0,C 180,E1 -5486.043,E2 -5486.043} C_VEL
LIN {X 0,Y 509.2,Z 554.806,A -85,B 0,C 180,E1 -5486.835,E2 -5486.835} C_VEL
LIN {X 0,Y 509.189,Z 556.206,A -85,B 0,C 180,E1 -5487.626,E2 -5487.626} C_VEL
LIN {X 0,Y 509.073,Z 557.814,A -85,B 0,C 180,E1 -5489.208,E2 -5489.208} C_VEL
LIN {X 0,Y 509.069,Z 558.033,A -85,B 0,C 180,E1 -5489.999,E2 -5489.999} C_VEL
LIN {X 0,Y 509.112,Z 557.213,A -85,B 0,C 180,E1 -5491.581,E2 -5491.581} C_VEL
LIN {X 0,Y 509.189,Z 556.22,A -85,B 0,C 180,E1 -5492.373,E2 -5492.373} C_VEL
LIN {X 0,Y 509.2,Z 554.823,A -85,B 0,C 180,E1 -5493.164,E2 -5493.164} C_VEL
LIN {X 0,Y 509.204,Z 551.883,A -85,B 0,C 180,E1 -5494.353,E2 -5494.353} C_VEL
LIN {X 0,Y 509.292,Z 547.904,A -85,B 0,C 180,E1 -5495.543,E2 -5495.543} C_VEL
LIN {X 0,Y 509.372,Z 542.236,A -85,B 0,C 180,E1 -5496.844,E2 -5496.844} C_VEL
LIN {X 0,Y 509.543,Z 535.092,A -85,B 0,C 180,E1 -5498.127,E2 -5498.127} C_VEL
LIN {X 0,Y 509.755,Z 526.792,A -85,B 0,C 180,E1 -5499.322,E2 -5499.322} C_VEL
LIN {X 0,Y 510.011,Z 518.285,A -85,B 0,C 180,E1 -5500.319,E2 -5500.319} C_VEL
LIN {X 0,Y 510.392,Z 507.777,A -85,B 0,C 180,E1 -5501.315,E2 -5501.315} C_VEL
LIN {X 0,Y 510.708,Z 496.307,A -85,B 0,C 180,E1 -5502.189,E2 -5502.189} C_VEL
LIN {X 0,Y 510.994,Z 485.982,A -85,B 0,C 180,E1 -5502.813,E2 -5502.813} C_VEL
LIN {X 0,Y 511.279,Z 474.275,A -85,B 0,C 180,E1 -5503.361,E2 -5503.361} C_VEL
LIN {X 0,Y 511.547,Z 460.79,A -85,B 0,C 180,E1 -5503.81,E2 -5503.81} C_VEL
LIN {X 0,Y 511.801,Z 447.405,A -85,B 0,C 180,E1 -5504.081,E2 -5504.081} C_VEL
LIN {X 0,Y 512.111,Z 357.147,A -85,B 0,C 180,E1 -5505.357,E2 -5505.357} C_VEL
LIN {X 0,Y 510.246,Z 345.16,A -85,B 0,C 180,E1 -5505.587,E2 -5505.587} C_VEL
LIN {X 0,Y 510.748,Z 325.588,A -85,B 0,C 180,E1 -5508.658,E2 -5508.658} C_VEL
LIN {X 0,Y 511.243,Z 307.213,A -85,B 0,C 180,E1 -5511.575,E2 -5511.575} C_VEL
LIN {X 0,Y 511.467,Z 295.372,A -85,B 0,C 180,E1 -5513.483,E2 -5513.483} C_VEL
LIN {X 0,Y 509.907,Z 286.97,A -85,B 0,C 180,E1 -5514.954,E2 -5514.954} C_VEL
LIN {X 0,Y 509.897,Z 286.974,A -85,B 0,C 180,E1 -5518.1,E2 -5518.1} C_VEL
LIN {X 0,Y 509.843,Z 286.971,A -85,B 0,C 180,E1 -5521.279,E2 -5521.279} C_VEL
LIN {X 0,Y 509.856,Z 286.979,A -85,B 0,C 180,E1 -5524.202,E2 -5524.202} C_VEL
LIN {X 0,Y 509.815,Z 286.974,A -85,B 0,C 180,E1 -5527.34,E2 -5527.34} C_VEL
LIN {X 0,Y 509.834,Z 286.982,A -85,B 0,C 180,E1 -5530.381,E2 -5530.381} C_VEL
LIN {X 0,Y 509.819,Z 286.975,A -85,B 0,C 180,E1 -5533.061,E2 -5533.061} C_VEL
LIN {X 0,Y 509.825,Z 286.974,A -85,B 0,C 180,E1 -5535.791,E2 -5535.791} C_VEL
LIN {X 0,Y 509.853,Z 286.98,A -85,B 0,C 180,E1 -5538.574,E2 -5538.574} C_VEL
LIN {X 0,Y 509.846,Z 286.97,A -85,B 0,C 180,E1 -5541.785,E2 -5541.785} C_VEL
LIN {X 0,Y 509.835,Z 286.98,A -85,B 0,C 180,E1 -5544.622,E2 -5544.622} C_VEL
LIN {X 0,Y 509.858,Z 286.97,A -85,B 0,C 180,E1 -5547.481,E2 -5547.481} C_VEL
LIN {X 0,Y 509.873,Z 286.968,A -85,B 0,C 180,E1 -5550.268,E2 -5550.268} C_VEL
LIN {X 0,Y 509.879,Z 286.976,A -85,B 0,C 180,E1 -5552.944,E2 -5552.944} C_VEL
LIN {X 0,Y 509.862,Z 286.971,A -85,B 0,C 180,E1 -5555.574,E2 -5555.574} C_VEL
LIN {X 0,Y 509.841,Z 286.979,A -85,B 0,C 180,E1 -5558.998,E2 -5558.998} C_VEL
LIN {X 0,Y 509.879,Z 286.967,A -85,B 0,C 180,E1 -5561.999,E2 -5561.999} C_VEL
LIN {X 0,Y 509.901,Z 286.967,A -85,B 0,C 180,E1 -5564.818,E2 -5564.818} C_VEL
LIN {X 0,Y 509.896,Z 286.965,A -85,B 0,C 180,E1 -5568.121,E2 -5568.121} C_VEL
LIN {X 0,Y 509.909,Z 286.97,A -85,B 0,C 180,E1 -5571.28,E2 -5571.28} C_VEL
LIN {X 0,Y 509.968,Z 286.962,A -85,B 0,C 180,E1 -5573.67,E2 -5573.67} C_VEL
LIN {X 0,Y 510.043,Z 286.956,A -85,B 0,C 180,E1 -5577.631,E2 -5577.631} C_VEL
LIN {X 0,Y 510.044,Z 286.95,A -85,B 0,C 180,E1 -5580,E2 -5580} C_VEL
LIN {X 0,Y 510.043,Z 286.947,A -85,B 0,C 180,E1 -5582.369,E2 -5582.369} C_VEL
LIN {X 0,Y 509.965,Z 286.961,A -85,B 0,C 180,E1 -5585.536,E2 -5585.536} C_VEL
LIN {X 0,Y 509.905,Z 286.963,A -85,B 0,C 180,E1 -5588.72,E2 -5588.72} C_VEL
LIN {X 0,Y 509.894,Z 286.973,A -85,B 0,C 180,E1 -5591.932,E2 -5591.932} C_VEL
LIN {X 0,Y 509.884,Z 286.966,A -85,B 0,C 180,E1 -5595.242,E2 -5595.242} C_VEL
LIN {X 0,Y 509.879,Z 286.974,A -85,B 0,C 180,E1 -5598.001,E2 -5598.001} C_VEL
LIN {X 0,Y 509.84,Z 286.972,A -85,B 0,C 180,E1 -5601.002,E2 -5601.002} C_VEL
LIN {X 0,Y 509.813,Z 286.975,A -85,B 0,C 180,E1 -5603.564,E2 -5603.564} C_VEL
LIN {X 0,Y 509.877,Z 286.977,A -85,B 0,C 180,E1 -5606.373,E2 -5606.373} C_VEL
LIN {X 0,Y 509.863,Z 286.972,A -85,B 0,C 180,E1 -5608.845,E2 -5608.845} C_VEL
LIN {X 0,Y 509.811,Z 286.975,A -85,B 0,C 180,E1 -5611.591,E2 -5611.591} C_VEL
LIN {X 0,Y 509.839,Z 286.978,A -85,B 0,C 180,E1 -5614.415,E2 -5614.415} C_VEL
LIN {X 0,Y 509.809,Z 286.976,A -85,B 0,C 180,E1 -5617.342,E2 -5617.342} C_VEL
LIN {X 0,Y 509.811,Z 286.979,A -85,B 0,C 180,E1 -5620.385,E2 -5620.385} C_VEL
LIN {X 0,Y 509.794,Z 286.983,A -85,B 0,C 180,E1 -5623.06,E2 -5623.06} C_VEL
LIN {X 0,Y 509.816,Z 286.974,A -85,B 0,C 180,E1 -5625.794,E2 -5625.794} C_VEL
LIN {X 0,Y 509.827,Z 286.977,A -85,B 0,C 180,E1 -5628.573,E2 -5628.573} C_VEL
LIN {X 0,Y 509.844,Z 286.971,A -85,B 0,C 180,E1 -5631.788,E2 -5631.788} C_VEL
LIN {X 0,Y 509.802,Z 286.977,A -85,B 0,C 180,E1 -5633.719,E2 -5633.719} C_VEL
LIN {X 0,Y 509.142,Z 287.059,A -85,B 0,C 180,E1 -5634.379,E2 -5634.379} C_VEL
LIN {X 0,Y 506.338,Z 287.412,A -85,B 0,C 180,E1 -5635.451,E2 -5635.451} C_VEL
LIN {X 0,Y 503.952,Z 287.713,A -85,B 0,C 180,E1 -5636.315,E2 -5636.315} C_VEL
LIN {X 0,Y 502.903,Z 287.842,A -85,B 0,C 180,E1 -5636.981,E2 -5636.981} C_VEL
LIN {X 0,Y 502.804,Z 287.851,A -85,B 0,C 180,E1 -5637.207,E2 -5637.207} C_VEL
LIN {X 0,Y 502.807,Z 287.848,A -85,B 0,C 180,E1 -5640.067,E2 -5640.067} C_VEL
LIN {X 0,Y 502.77,Z 287.86,A -85,B 0,C 180,E1 -5643.461,E2 -5643.461} C_VEL
LIN {X 0,Y 502.764,Z 287.854,A -85,B 0,C 180,E1 -5646.086,E2 -5646.086} C_VEL
LIN {X 0,Y 502.783,Z 287.851,A -85,B 0,C 180,E1 -5648.69,E2 -5648.69} C_VEL
LIN {X 0,Y 502.811,Z 287.851,A -85,B 0,C 180,E1 -5651.248,E2 -5651.248} C_VEL
LIN {X 0,Y 502.838,Z 287.843,A -85,B 0,C 180,E1 -5654.665,E2 -5654.665} C_VEL
LIN {X 0,Y 502.84,Z 287.848,A -85,B 0,C 180,E1 -5658.061,E2 -5658.061} C_VEL
LIN {X 0,Y 502.834,Z 287.848,A -85,B 0,C 180,E1 -5661.157,E2 -5661.157} C_VEL
LIN {X 0,Y 502.926,Z 288.032,A -85,B 0,C 180,E1 -5664.035,E2 -5664.035} C_VEL
LIN {X 0,Y 503.439,Z 292.88,A -85,B 0,C 180,E1 -5664.995,E2 -5664.995} C_VEL
LIN {X 0,Y 503.271,Z 306.409,A -85,B 0,C 180,E1 -5667.6,E2 -5667.6} C_VEL
LIN {X 0,Y 503.181,Z 309.821,A -85,B 0,C 180,E1 -5668.25,E2 -5668.25} C_VEL
LIN {X 0,Y 505.424,Z 321.482,A -85,B 0,C 180,E1 -5668.494,E2 -5668.494} C_VEL
LIN {X 0,Y 504.922,Z 416.721,A -85,B 0,C 180,E1 -5669.876,E2 -5669.876} C_VEL
LIN {X 0,Y 504.661,Z 429.128,A -85,B 0,C 180,E1 -5670.2,E2 -5670.2} C_VEL
LIN {X 0,Y 504.409,Z 441.877,A -85,B 0,C 180,E1 -5670.699,E2 -5670.699} C_VEL
LIN {X 0,Y 504.132,Z 453.219,A -85,B 0,C 180,E1 -5671.299,E2 -5671.299} C_VEL
LIN {X 0,Y 503.741,Z 464.9,A -85,B 0,C 180,E1 -5672.099,E2 -5672.099} C_VEL
LIN {X 0,Y 503.358,Z 475.368,A -85,B 0,C 180,E1 -5673.002,E2 -5673.002} C_VEL
LIN {X 0,Y 503.007,Z 484.827,A -85,B 0,C 180,E1 -5674.006,E2 -5674.006} C_VEL
LIN {X 0,Y 502.71,Z 493.943,A -85,B 0,C 180,E1 -5675.214,E2 -5675.214} C_VEL
LIN {X 0,Y 502.542,Z 501.283,A -85,B 0,C 180,E1 -5676.424,E2 -5676.424} C_VEL
LIN {X 0,Y 502.344,Z 507.205,A -85,B 0,C 180,E1 -5677.638,E2 -5677.638} C_VEL
LIN {X 0,Y 502.219,Z 511.889,A -85,B 0,C 180,E1 -5678.855,E2 -5678.855} C_VEL
LIN {X 0,Y 502.181,Z 515.466,A -85,B 0,C 180,E1 -5680.075,E2 -5680.075} C_VEL
LIN {X 0,Y 502.111,Z 518.432,A -85,B 0,C 180,E1 -5681.539,E2 -5681.539} C_VEL
LIN {X 0,Y 501.999,Z 519.978,A -85,B 0,C 180,E1 -5682.945,E2 -5682.945} C_VEL
LIN {X 0,Y 502.008,Z 520.321,A -85,B 0,C 180,E1 -5683.769,E2 -5683.769} C_VEL
LIN {X 0,Y 502.025,Z 520.072,A -85,B 0,C 180,E1 -5684.993,E2 -5684.993} C_VEL
LIN {X 0,Y 501.993,Z 518.849,A -85,B 0,C 180,E1 -5686.261,E2 -5686.261} C_VEL
LIN {X 0,Y 502.055,Z 517.498,A -85,B 0,C 180,E1 -5687.096,E2 -5687.096} C_VEL
LIN {X 0,Y 502.162,Z 514.592,A -85,B 0,C 180,E1 -5688.355,E2 -5688.355} C_VEL
LIN {X 0,Y 502.281,Z 510.554,A -85,B 0,C 180,E1 -5689.622,E2 -5689.622} C_VEL
LIN {X 0,Y 502.397,Z 505.237,A -85,B 0,C 180,E1 -5690.899,E2 -5690.899} C_VEL
LIN {X 0,Y 502.589,Z 498.388,A -85,B 0,C 180,E1 -5692.183,E2 -5692.183} C_VEL
LIN {X 0,Y 502.878,Z 491.326,A -85,B 0,C 180,E1 -5693.254,E2 -5693.254} C_VEL
LIN {X 0,Y 503.144,Z 482.664,A -85,B 0,C 180,E1 -5694.335,E2 -5694.335} C_VEL
LIN {X 0,Y 503.426,Z 473.426,A -85,B 0,C 180,E1 -5695.278,E2 -5695.278} C_VEL
LIN {X 0,Y 503.808,Z 462.486,A -85,B 0,C 180,E1 -5696.178,E2 -5696.178} C_VEL
LIN {X 0,Y 504.227,Z 450.568,A -85,B 0,C 180,E1 -5696.947,E2 -5696.947} C_VEL
LIN {X 0,Y 504.474,Z 438.669,A -85,B 0,C 180,E1 -5697.539,E2 -5697.539} C_VEL
LIN {X 0,Y 504.679,Z 425.946,A -85,B 0,C 180,E1 -5697.992,E2 -5697.992} C_VEL
LIN {X 0,Y 504.885,Z 412.894,A -85,B 0,C 180,E1 -5698.285,E2 -5698.285} C_VEL
LIN {X 0,Y 505.452,Z 321.689,A -85,B 0,C 180,E1 -5699.595,E2 -5699.595} C_VEL
LIN {X 0,Y 503.224,Z 309.611,A -85,B 0,C 180,E1 -5699.863,E2 -5699.863} C_VEL
LIN {X 0,Y 503.457,Z 294.006,A -85,B 0,C 180,E1 -5702.747,E2 -5702.747} C_VEL
LIN {X 0,Y 503.02,Z 288.74,A -85,B 0,C 180,E1 -5703.744,E2 -5703.744} C_VEL
LIN {X 0,Y 502.853,Z 287.851,A -85,B 0,C 180,E1 -5703.932,E2 -5703.932} C_VEL
LIN {X 0,Y 502.78,Z 287.852,A -85,B 0,C 180,E1 -5707.178,E2 -5707.178} C_VEL
LIN {X 0,Y 502.79,Z 287.855,A -85,B 0,C 180,E1 -5710.015,E2 -5710.015} C_VEL
LIN {X 0,Y 502.805,Z 287.855,A -85,B 0,C 180,E1 -5712.199,E2 -5712.199} C_VEL
LIN {X 0,Y 502.787,Z 287.853,A -85,B 0,C 180,E1 -5715.47,E2 -5715.47} C_VEL
LIN {X 0,Y 502.821,Z 287.852,A -85,B 0,C 180,E1 -5718.934,E2 -5718.934} C_VEL
LIN {X 0,Y 502.794,Z 287.85,A -85,B 0,C 180,E1 -5722.046,E2 -5722.046} C_VEL
LIN {X 0,Y 502.8,Z 287.856,A -85,B 0,C 180,E1 -5725.034,E2 -5725.034} C_VEL
LIN {X 0,Y 502.784,Z 287.851,A -85,B 0,C 180,E1 -5727.915,E2 -5727.915} C_VEL
LIN {X 0,Y 502.825,Z 287.848,A -85,B 0,C 180,E1 -5730.712,E2 -5730.712} C_VEL
LIN {X 0,Y 502.863,Z 287.845,A -85,B 0,C 180,E1 -5733.439,E2 -5733.439} C_VEL
LIN {X 0,Y 502.786,Z 287.85,A -85,B 0,C 180,E1 -5736.086,E2 -5736.086} C_VEL
LIN {X 0,Y 502.783,Z 287.852,A -85,B 0,C 180,E1 -5738.689,E2 -5738.689} C_VEL
LIN {X 0,Y 502.829,Z 287.85,A -85,B 0,C 180,E1 -5741.248,E2 -5741.248} C_VEL
LIN {X 0,Y 502.821,Z 287.85,A -85,B 0,C 180,E1 -5743.767,E2 -5743.767} C_VEL
LIN {X 0,Y 502.83,Z 287.844,A -85,B 0,C 180,E1 -5746.255,E2 -5746.255} C_VEL
LIN {X 0,Y 502.876,Z 287.839,A -85,B 0,C 180,E1 -5748.717,E2 -5748.717} C_VEL
LIN {X 0,Y 502.901,Z 287.842,A -85,B 0,C 180,E1 -5751.967,E2 -5751.967} C_VEL
LIN {X 0,Y 502.931,Z 287.832,A -85,B 0,C 180,E1 -5754.386,E2 -5754.386} C_VEL
LIN {X 0,Y 503.023,Z 287.824,A -85,B 0,C 180,E1 -5757.598,E2 -5757.598} C_VEL
LIN {X 0,Y 503.027,Z 287.824,A -85,B 0,C 180,E1 -5760,E2 -5760} C_VEL
LIN {X 0,Y 503.024,Z 287.824,A -85,B 0,C 180,E1 -5762.402,E2 -5762.402} C_VEL
LIN {X 0,Y 502.931,Z 287.832,A -85,B 0,C 180,E1 -5765.614,E2 -5765.614} C_VEL
LIN {X 0,Y 502.9,Z 287.84,A -85,B 0,C 180,E1 -5768.033,E2 -5768.033} C_VEL
LIN {X 0,Y 502.876,Z 287.834,A -85,B 0,C 180,E1 -5771.283,E2 -5771.283} C_VEL
LIN {X 0,Y 502.844,Z 287.848,A -85,B 0,C 180,E1 -5774.571,E2 -5774.571} C_VEL
LIN {X 0,Y 502.855,Z 287.842,A -85,B 0,C 180,E1 -5777.907,E2 -5777.907} C_VEL
LIN {X 0,Y 502.829,Z 287.851,A -85,B 0,C 180,E1 -5780.536,E2 -5780.536} C_VEL
LIN {X 0,Y 502.791,Z 287.854,A -85,B 0,C 180,E1 -5783.041,E2 -5783.041} C_VEL
LIN {X 0,Y 502.84,Z 287.84,A -85,B 0,C 180,E1 -5785.676,E2 -5785.676} C_VEL
LIN {X 0,Y 502.84,Z 287.846,A -85,B 0,C 180,E1 -5788.373,E2 -5788.373} C_VEL
LIN {X 0,Y 502.793,Z 287.852,A -85,B 0,C 180,E1 -5791.499,E2 -5791.499} C_VEL
LIN {X 0,Y 502.789,Z 287.847,A -85,B 0,C 180,E1 -5793.995,E2 -5793.995} C_VEL
LIN {X 0,Y 502.778,Z 287.858,A -85,B 0,C 180,E1 -5797.178,E2 -5797.178} C_VEL
LIN {X 0,Y 502.789,Z 287.85,A -85,B 0,C 180,E1 -5800.015,E2 -5800.015} C_VEL
LIN {X 0,Y 502.804,Z 287.849,A -85,B 0,C 180,E1 -5802.199,E2 -5802.199} C_VEL
LIN {X 0,Y 502.787,Z 287.858,A -85,B 0,C 180,E1 -5805.47,E2 -5805.47} C_VEL
LIN {X 0,Y 502.821,Z 287.848,A -85,B 0,C 180,E1 -5808.934,E2 -5808.934} C_VEL
LIN {X 0,Y 502.795,Z 287.855,A -85,B 0,C 180,E1 -5812.046,E2 -5812.046} C_VEL
LIN {X 0,Y 502.801,Z 287.85,A -85,B 0,C 180,E1 -5815.034,E2 -5815.034} C_VEL
LIN {X 0,Y 502.786,Z 287.859,A -85,B 0,C 180,E1 -5817.915,E2 -5817.915} C_VEL
LIN {X 0,Y 502.826,Z 287.848,A -85,B 0,C 180,E1 -5820.712,E2 -5820.712} C_VEL
LIN {X 0,Y 502.866,Z 287.847,A -85,B 0,C 180,E1 -5823.439,E2 -5823.439} C_VEL
LIN {X 0,Y 502.869,Z 287.941,A -85,B 0,C 180,E1 -5824.952,E2 -5824.952} C_VEL
LIN {X 0,Y 504.506,Z 297.154,A -85,B 0,C 180,E1 -5826.559,E2 -5826.559} C_VEL
LIN {X 0,Y 504.145,Z 312.01,A -85,B 0,C 180,E1 -5828.975,E2 -5828.975} C_VEL
LIN {X 0,Y 503.588,Z 331.671,A -85,B 0,C 180,E1 -5832.119,E2 -5832.119} C_VEL
LIN {X 0,Y 503.235,Z 344.897,A -85,B 0,C 180,E1 -5834.192,E2 -5834.192} C_VEL
LIN {X 0,Y 505.319,Z 359.951,A -85,B 0,C 180,E1 -5834.477,E2 -5834.477} C_VEL
LIN {X 0,Y 504.822,Z 452.898,A -85,B 0,C 180,E1 -5835.822,E2 -5835.822} C_VEL
LIN {X 0,Y 504.532,Z 466.289,A -85,B 0,C 180,E1 -5836.173,E2 -5836.173} C_VEL
LIN {X 0,Y 504.216,Z 479.65,A -85,B 0,C 180,E1 -5836.703,E2 -5836.703} C_VEL
LIN {X 0,Y 503.875,Z 491.926,A -85,B 0,C 180,E1 -5837.378,E2 -5837.378} C_VEL
LIN {X 0,Y 503.538,Z 503.798,A -85,B 0,C 180,E1 -5838.221,E2 -5838.221} C_VEL
LIN {X 0,Y 503.182,Z 514.032,A -85,B 0,C 180,E1 -5839.131,E2 -5839.131} C_VEL
LIN {X 0,Y 502.834,Z 523.237,A -85,B 0,C 180,E1 -5840.141,E2 -5840.141} C_VEL
LIN {X 0,Y 502.556,Z 532.208,A -85,B 0,C 180,E1 -5841.353,E2 -5841.353} C_VEL
LIN {X 0,Y 502.347,Z 539.431,A -85,B 0,C 180,E1 -5842.564,E2 -5842.564} C_VEL
LIN {X 0,Y 502.236,Z 544.306,A -85,B 0,C 180,E1 -5843.572,E2 -5843.572} C_VEL
LIN {X 0,Y 502.174,Z 549.047,A -85,B 0,C 180,E1 -5844.78,E2 -5844.78} C_VEL
LIN {X 0,Y 502.139,Z 552.67,A -85,B 0,C 180,E1 -5845.987,E2 -5845.987} C_VEL
LIN {X 0,Y 502.12,Z 554.539,A -85,B 0,C 180,E1 -5846.79,E2 -5846.79} C_VEL
LIN {X 0,Y 502.091,Z 555.94,A -85,B 0,C 180,E1 -5847.593,E2 -5847.593} C_VEL
LIN {X 0,Y 501.99,Z 557.55,A -85,B 0,C 180,E1 -5849.197,E2 -5849.197} C_VEL
LIN {X 0,Y 501.983,Z 557.769,A -85,B 0,C 180,E1 -5849.999,E2 -5849.999} C_VEL
LIN {X 0,Y 502.036,Z 556.95,A -85,B 0,C 180,E1 -5851.604,E2 -5851.604} C_VEL
LIN {X 0,Y 502.091,Z 555.956,A -85,B 0,C 180,E1 -5852.406,E2 -5852.406} C_VEL
LIN {X 0,Y 502.12,Z 554.56,A -85,B 0,C 180,E1 -5853.209,E2 -5853.209} C_VEL
LIN {X 0,Y 502.102,Z 551.618,A -85,B 0,C 180,E1 -5854.415,E2 -5854.415} C_VEL
LIN {X 0,Y 502.208,Z 547.639,A -85,B 0,C 180,E1 -5855.621,E2 -5855.621} C_VEL
LIN {X 0,Y 502.323,Z 541.617,A -85,B 0,C 180,E1 -5857.011,E2 -5857.011} C_VEL
LIN {X 0,Y 502.476,Z 534.825,A -85,B 0,C 180,E1 -5858.242,E2 -5858.242} C_VEL
LIN {X 0,Y 502.715,Z 526.524,A -85,B 0,C 180,E1 -5859.454,E2 -5859.454} C_VEL
LIN {X 0,Y 502.988,Z 518.015,A -85,B 0,C 180,E1 -5860.465,E2 -5860.465} C_VEL
LIN {X 0,Y 503.416,Z 507.505,A -85,B 0,C 180,E1 -5861.474,E2 -5861.474} C_VEL
LIN {X 0,Y 503.736,Z 496.032,A -85,B 0,C 180,E1 -5862.36,E2 -5862.36} C_VEL
LIN {X 0,Y 504.047,Z 485.704,A -85,B 0,C 180,E1 -5862.992,E2 -5862.992} C_VEL
LIN {X 0,Y 504.359,Z 473.991,A -85,B 0,C 180,E1 -5863.548,E2 -5863.548} C_VEL
LIN {X 0,Y 504.675,Z 460.498,A -85,B 0,C 180,E1 -5864.002,E2 -5864.002} C_VEL
LIN {X 0,Y 504.91,Z 447.085,A -85,B 0,C 180,E1 -5864.278,E2 -5864.278} C_VEL
LIN {X 0,Y 505.294,Z 358.158,A -85,B 0,C 180,E1 -5865.551,E2 -5865.551} C_VEL
LIN {X 0,Y 503.246,Z 344.82,A -85,B 0,C 180,E1 -5865.823,E2 -5865.823} C_VEL
LIN {X 0,Y 503.778,Z 325.312,A -85,B 0,C 180,E1 -5868.925,E2 -5868.925} C_VEL
LIN {X 0,Y 504.378,Z 305.617,A -85,B 0,C 180,E1 -5872.099,E2 -5872.099} C_VEL
LIN {X 0,Y 504.565,Z 297.347,A -85,B 0,C 180,E1 -5873.446,E2 -5873.446} C_VEL
LIN {X 0,Y 502.872,Z 287.847,A -85,B 0,C 180,E1 -5875.107,E2 -5875.107} C_VEL
LIN {X 0,Y 502.843,Z 287.851,A -85,B 0,C 180,E1 -5878.294,E2 -5878.294} C_VEL
LIN {X 0,Y 502.79,Z 287.851,A -85,B 0,C 180,E1 -5881.498,E2 -5881.498} C_VEL
LIN {X 0,Y 502.801,Z 287.854,A -85,B 0,C 180,E1 -5884.443,E2 -5884.443} C_VEL
LIN {X 0,Y 502.777,Z 287.851,A -85,B 0,C 180,E1 -5887.177,E2 -5887.177} C_VEL
LIN {X 0,Y 502.783,Z 287.855,A -85,B 0,C 180,E1 -5890.014,E2 -5890.014} C_VEL
LIN {X 0,Y 502.798,Z 287.855,A -85,B 0,C 180,E1 -5892.198,E2 -5892.198} C_VEL
LIN {X 0,Y 502.795,Z 287.849,A -85,B 0,C 180,E1 -5895.467,E2 -5895.467} C_VEL
LIN {X 0,Y 502.824,Z 287.846,A -85,B 0,C 180,E1 -5897.863,E2 -5897.863} C_VEL
LIN {X 0,Y 502.796,Z 287.852,A -85,B 0,C 180,E1 -5901.023,E2 -5901.023} C_VEL
LIN {X 0,Y 502.776,Z 287.853,A -85,B 0,C 180,E1 -5904.167,E2 -5904.167} C_VEL
LIN {X 0,Y 502.825,Z 287.852,A -85,B 0,C 180,E1 -5906.992,E2 -5906.992} C_VEL
LIN {X 0,Y 502.822,Z 287.846,A -85,B 0,C 180,E1 -5910.061,E2 -5910.061} C_VEL
LIN {X 0,Y 502.827,Z 287.848,A -85,B 0,C 180,E1 -5912.533,E2 -5912.533} C_VEL
LIN {X 0,Y 502.82,Z 287.851,A -85,B 0,C 180,E1 -5915.298,E2 -5915.298} C_VEL
LIN {X 0,Y 502.772,Z 287.852,A -85,B 0,C 180,E1 -5917.826,E2 -5917.826} C_VEL
LIN {X 0,Y 502.815,Z 287.847,A -85,B 0,C 180,E1 -5920.4,E2 -5920.4} C_VEL
LIN {X 0,Y 502.824,Z 287.85,A -85,B 0,C 180,E1 -5922.931,E2 -5922.931} C_VEL
LIN {X 0,Y 502.842,Z 287.85,A -85,B 0,C 180,E1 -5925.429,E2 -5925.429} C_VEL
LIN {X 0,Y 502.871,Z 287.84,A -85,B 0,C 180,E1 -5928.717,E2 -5928.717} C_VEL
LIN {X 0,Y 502.893,Z 287.839,A -85,B 0,C 180,E1 -5931.967,E2 -5931.967} C_VEL
LIN {X 0,Y 502.928,Z 287.832,A -85,B 0,C 180,E1 -5934.386,E2 -5934.386} C_VEL
LIN {X 0,Y 503.014,Z 287.831,A -85,B 0,C 180,E1 -5937.598,E2 -5937.598} C_VEL
LIN {X 0,Y 503.015,Z 287.826,A -85,B 0,C 180,E1 -5940,E2 -5940} C_VEL
LIN {X 0,Y 503.014,Z 287.823,A -85,B 0,C 180,E1 -5942.402,E2 -5942.402} C_VEL
LIN {X 0,Y 502.918,Z 287.84,A -85,B 0,C 180,E1 -5945.614,E2 -5945.614} C_VEL
LIN {X 0,Y 502.864,Z 287.84,A -85,B 0,C 180,E1 -5948.844,E2 -5948.844} C_VEL
LIN {X 0,Y 502.836,Z 287.852,A -85,B 0,C 180,E1 -5952.102,E2 -5952.102} C_VEL
LIN {X 0,Y 502.839,Z 287.844,A -85,B 0,C 180,E1 -5955.4,E2 -5955.4} C_VEL
LIN {X 0,Y 502.836,Z 287.853,A -85,B 0,C 180,E1 -5958.123,E2 -5958.123} C_VEL
LIN {X 0,Y 502.82,Z 287.85,A -85,B 0,C 180,E1 -5960.537,E2 -5960.537} C_VEL
LIN {X 0,Y 502.779,Z 287.851,A -85,B 0,C 180,E1 -5963.041,E2 -5963.041} C_VEL
LIN {X 0,Y 502.793,Z 287.85,A -85,B 0,C 180,E1 -5965.678,E2 -5965.678} C_VEL
LIN {X 0,Y 502.827,Z 287.854,A -85,B 0,C 180,E1 -5968.374,E2 -5968.374} C_VEL
LIN {X 0,Y 502.784,Z 287.85,A -85,B 0,C 180,E1 -5971.499,E2 -5971.499} C_VEL
LIN {X 0,Y 502.795,Z 287.85,A -85,B 0,C 180,E1 -5973.995,E2 -5973.995} C_VEL
LIN {X 0,Y 502.77,Z 287.854,A -85,B 0,C 180,E1 -5977.178,E2 -5977.178} C_VEL
LIN {X 0,Y 502.766,Z 287.853,A -85,B 0,C 180,E1 -5980.018,E2 -5980.018} C_VEL
LIN {X 0,Y 502.797,Z 287.85,A -85,B 0,C 180,E1 -5982.2,E2 -5982.2} C_VEL
LIN {X 0,Y 502.78,Z 287.852,A -85,B 0,C 180,E1 -5985.471,E2 -5985.471} C_VEL
LIN {X 0,Y 502.79,Z 287.849,A -85,B 0,C 180,E1 -5987.862,E2 -5987.862} C_VEL
LIN {X 0,Y 502.788,Z 287.859,A -85,B 0,C 180,E1 -5991.024,E2 -5991.024} C_VEL
LIN {X 0,Y 502.767,Z 287.852,A -85,B 0,C 180,E1 -5994.171,E2 -5994.171} C_VEL
LIN {X 0,Y 502.804,Z 287.851,A -85,B 0,C 180,E1 -5997.207,E2 -5997.207} C_VEL
LIN {X 0,Y 502.101,Z 287.938,A -85,B 0,C 180,E1 -5997.875,E2 -5997.875} C_VEL
LIN {X 0,Y 499.24,Z 288.297,A -85,B 0,C 180,E1 -5998.961,E2 -5998.961} C_VEL
LIN {X 0,Y 496.84,Z 288.592,A -85,B 0,C 180,E1 -5999.836,E2 -5999.836} C_VEL
LIN {X 0,Y 495.808,Z 288.72,A -85,B 0,C 180,E1 -6000.511,E2 -6000.511} C_VEL
LIN {X 0,Y 495.722,Z 288.732,A -85,B 0,C 180,E1 -6000.74,E2 -6000.74} C_VEL
LIN {X 0,Y 495.71,Z 288.733,A -85,B 0,C 180,E1 -6003.929,E2 -6003.929} C_VEL
LIN {X 0,Y 495.757,Z 288.73,A -85,B 0,C 180,E1 -6007.141,E2 -6007.141} C_VEL
LIN {X 0,Y 495.767,Z 288.726,A -85,B 0,C 180,E1 -6010.11,E2 -6010.11} C_VEL
LIN {X 0,Y 495.742,Z 288.727,A -85,B 0,C 180,E1 -6012.681,E2 -6012.681} C_VEL
LIN {X 0,Y 495.778,Z 288.726,A -85,B 0,C 180,E1 -6015.218,E2 -6015.218} C_VEL
LIN {X 0,Y 495.79,Z 288.722,A -85,B 0,C 180,E1 -6018.554,E2 -6018.554} C_VEL
LIN {X 0,Y 495.811,Z 288.729,A -85,B 0,C 180,E1 -6021.852,E2 -6021.852} C_VEL
LIN {X 0,Y 495.873,Z 288.893,A -85,B 0,C 180,E1 -6023.899,E2 -6023.899} C_VEL
LIN {X 0,Y 496.456,Z 293.999,A -85,B 0,C 180,E1 -6024.925,E2 -6024.925} C_VEL
LIN {X 0,Y 496.284,Z 307.64,A -85,B 0,C 180,E1 -6027.566,E2 -6027.566} C_VEL
LIN {X 0,Y 496.187,Z 310.027,A -85,B 0,C 180,E1 -6028.022,E2 -6028.022} C_VEL
LIN {X 0,Y 498.56,Z 322.117,A -85,B 0,C 180,E1 -6028.284,E2 -6028.284} C_VEL
LIN {X 0,Y 498.053,Z 417.72,A -85,B 0,C 180,E1 -6029.697,E2 -6029.697} C_VEL
LIN {X 0,Y 497.745,Z 429.919,A -85,B 0,C 180,E1 -6030.026,E2 -6030.026} C_VEL
LIN {X 0,Y 497.496,Z 443.077,A -85,B 0,C 180,E1 -6030.557,E2 -6030.557} C_VEL
LIN {X 0,Y 497.144,Z 454.986,A -85,B 0,C 180,E1 -6031.216,E2 -6031.216} C_VEL
LIN {X 0,Y 496.757,Z 466.356,A -85,B 0,C 180,E1 -6032.028,E2 -6032.028} C_VEL
LIN {X 0,Y 496.373,Z 476.623,A -85,B 0,C 180,E1 -6032.943,E2 -6032.943} C_VEL
LIN {X 0,Y 496.026,Z 485.043,A -85,B 0,C 180,E1 -6033.86,E2 -6033.86} C_VEL
LIN {X 0,Y 495.685,Z 494.175,A -85,B 0,C 180,E1 -6035.084,E2 -6035.084} C_VEL
LIN {X 0,Y 495.499,Z 501.521,A -85,B 0,C 180,E1 -6036.311,E2 -6036.311} C_VEL
LIN {X 0,Y 495.325,Z 506.541,A -85,B 0,C 180,E1 -6037.337,E2 -6037.337} C_VEL
LIN {X 0,Y 495.172,Z 511.42,A -85,B 0,C 180,E1 -6038.571,E2 -6038.571} C_VEL
LIN {X 0,Y 495.081,Z 515.183,A -85,B 0,C 180,E1 -6039.809,E2 -6039.809} C_VEL
LIN {X 0,Y 495.048,Z 517.127,A -85,B 0,C 180,E1 -6040.636,E2 -6040.636} C_VEL
LIN {X 0,Y 495.01,Z 518.8,A -85,B 0,C 180,E1 -6041.58,E2 -6041.58} C_VEL
LIN {X 0,Y 494.921,Z 520.361,A -85,B 0,C 180,E1 -6043.133,E2 -6043.133} C_VEL
LIN {X 0,Y 494.916,Z 520.627,A -85,B 0,C 180,E1 -6043.97,E2 -6043.97} C_VEL
LIN {X 0,Y 494.942,Z 520.296,A -85,B 0,C 180,E1 -6045.076,E2 -6045.076} C_VEL
LIN {X 0,Y 494.91,Z 518.83,A -85,B 0,C 180,E1 -6046.5,E2 -6046.5} C_VEL
LIN {X 0,Y 495.067,Z 515.975,A -85,B 0,C 180,E1 -6047.984,E2 -6047.984} C_VEL
LIN {X 0,Y 495.184,Z 511.576,A -85,B 0,C 180,E1 -6049.483,E2 -6049.483} C_VEL
LIN {X 0,Y 495.35,Z 505.521,A -85,B 0,C 180,E1 -6050.993,E2 -6050.993} C_VEL
LIN {X 0,Y 495.573,Z 498.678,A -85,B 0,C 180,E1 -6052.294,E2 -6052.294} C_VEL
LIN {X 0,Y 495.878,Z 490.039,A -85,B 0,C 180,E1 -6053.602,E2 -6053.602} C_VEL
LIN {X 0,Y 496.241,Z 481.291,A -85,B 0,C 180,E1 -6054.668,E2 -6054.668} C_VEL
LIN {X 0,Y 496.556,Z 470.945,A -85,B 0,C 180,E1 -6055.687,E2 -6055.687} C_VEL
LIN {X 0,Y 497.041,Z 459.817,A -85,B 0,C 180,E1 -6056.562,E2 -6056.562} C_VEL
LIN {X 0,Y 497.396,Z 448.85,A -85,B 0,C 180,E1 -6057.246,E2 -6057.246} C_VEL
LIN {X 0,Y 497.643,Z 436.409,A -85,B 0,C 180,E1 -6057.835,E2 -6057.835} C_VEL
LIN {X 0,Y 497.875,Z 423.077,A -85,B 0,C 180,E1 -6058.279,E2 -6058.279} C_VEL
LIN {X 0,Y 498.043,Z 408.899,A -85,B 0,C 180,E1 -6058.556,E2 -6058.556} C_VEL
LIN {X 0,Y 498.566,Z 322.206,A -85,B 0,C 180,E1 -6059.815,E2 -6059.815} C_VEL
LIN {X 0,Y 496.283,Z 309.88,A -85,B 0,C 180,E1 -6060.087,E2 -6060.087} C_VEL
LIN {X 0,Y 496.507,Z 294.175,A -85,B 0,C 180,E1 -6063.022,E2 -6063.022} C_VEL
LIN {X 0,Y 495.805,Z 288.729,A -85,B 0,C 180,E1 -6064.08,E2 -6064.08} C_VEL
LIN {X 0,Y 495.731,Z 288.73,A -85,B 0,C 180,E1 -6067.562,E2 -6067.562} C_VEL
LIN {X 0,Y 495.768,Z 288.731,A -85,B 0,C 180,E1 -6070.7,E2 -6070.7} C_VEL
LIN {X 0,Y 495.73,Z 288.734,A -85,B 0,C 180,E1 -6074.002,E2 -6074.002} C_VEL
LIN {X 0,Y 495.727,Z 288.734,A -85,B 0,C 180,E1 -6077.117,E2 -6077.117} C_VEL
LIN {X 0,Y 495.76,Z 288.728,A -85,B 0,C 180,E1 -6079.953,E2 -6079.953} C_VEL
LIN {X 0,Y 495.729,Z 288.735,A -85,B 0,C 180,E1 -6082.553,E2 -6082.553} C_VEL
LIN {X 0,Y 495.779,Z 288.726,A -85,B 0,C 180,E1 -6085.457,E2 -6085.457} C_VEL
LIN {X 0,Y 495.756,Z 288.728,A -85,B 0,C 180,E1 -6088.364,E2 -6088.364} C_VEL
LIN {X 0,Y 495.788,Z 288.726,A -85,B 0,C 180,E1 -6091.507,E2 -6091.507} C_VEL
LIN {X 0,Y 495.791,Z 288.722,A -85,B 0,C 180,E1 -6093.932,E2 -6093.932} C_VEL
LIN {X 0,Y 495.76,Z 288.731,A -85,B 0,C 180,E1 -6097.139,E2 -6097.139} C_VEL
LIN {X 0,Y 495.771,Z 288.723,A -85,B 0,C 180,E1 -6100.109,E2 -6100.109} C_VEL
LIN {X 0,Y 495.781,Z 288.723,A -85,B 0,C 180,E1 -6102.681,E2 -6102.681} C_VEL
LIN {X 0,Y 495.79,Z 288.726,A -85,B 0,C 180,E1 -6105.217,E2 -6105.217} C_VEL
LIN {X 0,Y 495.851,Z 288.714,A -85,B 0,C 180,E1 -6108.555,E2 -6108.555} C_VEL
LIN {X 0,Y 495.872,Z 288.719,A -85,B 0,C 180,E1 -6111.852,E2 -6111.852} C_VEL
LIN {X 0,Y 495.888,Z 288.71,A -85,B 0,C 180,E1 -6114.306,E2 -6114.306} C_VEL
LIN {X 0,Y 495.992,Z 288.699,A -85,B 0,C 180,E1 -6117.564,E2 -6117.564} C_VEL
LIN {X 0,Y 495.982,Z 288.692,A -85,B 0,C 180,E1 -6120.812,E2 -6120.812} C_VEL
LIN {X 0,Y 495.993,Z 288.699,A -85,B 0,C 180,E1 -6122.436,E2 -6122.436} C_VEL
LIN {X 0,Y 495.887,Z 288.71,A -85,B 0,C 180,E1 -6125.694,E2 -6125.694} C_VEL
LIN {X 0,Y 495.872,Z 288.717,A -85,B 0,C 180,E1 -6128.148,E2 -6128.148} C_VEL
LIN {X 0,Y 495.851,Z 288.709,A -85,B 0,C 180,E1 -6131.445,E2 -6131.445} C_VEL
LIN {X 0,Y 495.79,Z 288.724,A -85,B 0,C 180,E1 -6134.783,E2 -6134.783} C_VEL
LIN {X 0,Y 495.781,Z 288.722,A -85,B 0,C 180,E1 -6137.319,E2 -6137.319} C_VEL
LIN {X 0,Y 495.77,Z 288.725,A -85,B 0,C 180,E1 -6139.89,E2 -6139.89} C_VEL
LIN {X 0,Y 495.76,Z 288.733,A -85,B 0,C 180,E1 -6142.861,E2 -6142.861} C_VEL
LIN {X 0,Y 495.791,Z 288.719,A -85,B 0,C 180,E1 -6146.068,E2 -6146.068} C_VEL
LIN {X 0,Y 495.773,Z 288.732,A -85,B 0,C 180,E1 -6148.815,E2 -6148.815} C_VEL
LIN {X 0,Y 495.755,Z 288.727,A -85,B 0,C 180,E1 -6151.725,E2 -6151.725} C_VEL
LIN {X 0,Y 495.762,Z 288.726,A -85,B 0,C 180,E1 -6154.693,E2 -6154.693} C_VEL
LIN {X 0,Y 495.73,Z 288.733,A -85,B 0,C 180,E1 -6157.562,E2 -6157.562} C_VEL
LIN {X 0,Y 495.767,Z 288.726,A -85,B 0,C 180,E1 -6160.7,E2 -6160.7} C_VEL
LIN {X 0,Y 495.729,Z 288.732,A -85,B 0,C 180,E1 -6164.002,E2 -6164.002} C_VEL
LIN {X 0,Y 495.727,Z 288.735,A -85,B 0,C 180,E1 -6167.117,E2 -6167.117} C_VEL
LIN {X 0,Y 495.76,Z 288.727,A -85,B 0,C 180,E1 -6169.953,E2 -6169.953} C_VEL
LIN {X 0,Y 495.73,Z 288.732,A -85,B 0,C 180,E1 -6172.553,E2 -6172.553} C_VEL
LIN {X 0,Y 495.78,Z 288.729,A -85,B 0,C 180,E1 -6175.457,E2 -6175.457} C_VEL
LIN {X 0,Y 495.758,Z 288.728,A -85,B 0,C 180,E1 -6178.364,E2 -6178.364} C_VEL
LIN {X 0,Y 495.79,Z 288.727,A -85,B 0,C 180,E1 -6181.507,E2 -6181.507} C_VEL
LIN {X 0,Y 495.822,Z 288.727,A -85,B 0,C 180,E1 -6184.61,E2 -6184.61} C_VEL
LIN {X 0,Y 495.857,Z 288.985,A -85,B 0,C 180,E1 -6184.78,E2 -6184.78} C_VEL
LIN {X 0,Y 497.597,Z 298.698,A -85,B 0,C 180,E1 -6186.506,E2 -6186.506} C_VEL
LIN {X 0,Y 497.191,Z 313.202,A -85,B 0,C 180,E1 -6188.898,E2 -6188.898} C_VEL
LIN {X 0,Y 496.569,Z 332.743,A -85,B 0,C 180,E1 -6192.071,E2 -6192.071} C_VEL
LIN {X 0,Y 496.243,Z 344.478,A -85,B 0,C 180,E1 -6193.955,E2 -6193.955} C_VEL
LIN {X 0,Y 498.482,Z 360.518,A -85,B 0,C 180,E1 -6194.268,E2 -6194.268} C_VEL
LIN {X 0,Y 497.954,Z 452.71,A -85,B 0,C 180,E1 -6195.622,E2 -6195.622} C_VEL
LIN {X 0,Y 497.644,Z 466.057,A -85,B 0,C 180,E1 -6195.978,E2 -6195.978} C_VEL
LIN {X 0,Y 497.293,Z 479.393,A -85,B 0,C 180,E1 -6196.515,E2 -6196.515} C_VEL
LIN {X 0,Y 496.932,Z 490.535,A -85,B 0,C 180,E1 -6197.126,E2 -6197.126} C_VEL
LIN {X 0,Y 496.586,Z 502.219,A -85,B 0,C 180,E1 -6197.95,E2 -6197.95} C_VEL
LIN {X 0,Y 496.204,Z 512.699,A -85,B 0,C 180,E1 -6198.873,E2 -6198.873} C_VEL
LIN {X 0,Y 495.848,Z 521.27,A -85,B 0,C 180,E1 -6199.795,E2 -6199.795} C_VEL
LIN {X 0,Y 495.564,Z 529.181,A -85,B 0,C 180,E1 -6200.819,E2 -6200.819} C_VEL
LIN {X 0,Y 495.342,Z 536.911,A -85,B 0,C 180,E1 -6202.048,E2 -6202.048} C_VEL
LIN {X 0,Y 495.164,Z 544.035,A -85,B 0,C 180,E1 -6203.48,E2 -6203.48} C_VEL
LIN {X 0,Y 495.106,Z 548.778,A -85,B 0,C 180,E1 -6204.705,E2 -6204.705} C_VEL
LIN {X 0,Y 495.033,Z 552.401,A -85,B 0,C 180,E1 -6205.929,E2 -6205.929} C_VEL
LIN {X 0,Y 495.042,Z 554.273,A -85,B 0,C 180,E1 -6206.744,E2 -6206.744} C_VEL
LIN {X 0,Y 494.998,Z 555.674,A -85,B 0,C 180,E1 -6207.558,E2 -6207.558} C_VEL
LIN {X 0,Y 494.962,Z 556.675,A -85,B 0,C 180,E1 -6208.372,E2 -6208.372} C_VEL
LIN {X 0,Y 494.901,Z 557.505,A -85,B 0,C 180,E1 -6209.999,E2 -6209.999} C_VEL
LIN {X 0,Y 494.962,Z 556.687,A -85,B 0,C 180,E1 -6211.627,E2 -6211.627} C_VEL
LIN {X 0,Y 494.997,Z 555.693,A -85,B 0,C 180,E1 -6212.441,E2 -6212.441} C_VEL
LIN {X 0,Y 495.041,Z 554.296,A -85,B 0,C 180,E1 -6213.255,E2 -6213.255} C_VEL
LIN {X 0,Y 495.007,Z 551.354,A -85,B 0,C 180,E1 -6214.478,E2 -6214.478} C_VEL
LIN {X 0,Y 495.124,Z 547.374,A -85,B 0,C 180,E1 -6215.702,E2 -6215.702} C_VEL
LIN {X 0,Y 495.253,Z 541.25,A -85,B 0,C 180,E1 -6217.132,E2 -6217.132} C_VEL
LIN {X 0,Y 495.424,Z 534.558,A -85,B 0,C 180,E1 -6218.36,E2 -6218.36} C_VEL
LIN {X 0,Y 495.678,Z 526.255,A -85,B 0,C 180,E1 -6219.589,E2 -6219.589} C_VEL
LIN {X 0,Y 495.983,Z 517.745,A -85,B 0,C 180,E1 -6220.614,E2 -6220.614} C_VEL
LIN {X 0,Y 496.436,Z 507.233,A -85,B 0,C 180,E1 -6221.638,E2 -6221.638} C_VEL
LIN {X 0,Y 496.784,Z 495.705,A -85,B 0,C 180,E1 -6222.54,E2 -6222.54} C_VEL
LIN {X 0,Y 497.14,Z 483.486,A -85,B 0,C 180,E1 -6223.28,E2 -6223.28} C_VEL
LIN {X 0,Y 497.542,Z 471.088,A -85,B 0,C 180,E1 -6223.841,E2 -6223.841} C_VEL
LIN {X 0,Y 497.79,Z 458.33,A -85,B 0,C 180,E1 -6224.251,E2 -6224.251} C_VEL
LIN {X 0,Y 498.041,Z 444.893,A -85,B 0,C 180,E1 -6224.505,E2 -6224.505} C_VEL
LIN {X 0,Y 498.444,Z 358.739,A -85,B 0,C 180,E1 -6225.755,E2 -6225.755} C_VEL
LIN {X 0,Y 496.252,Z 344.644,A -85,B 0,C 180,E1 -6226.035,E2 -6226.035} C_VEL
LIN {X 0,Y 496.837,Z 325.028,A -85,B 0,C 180,E1 -6229.2,E2 -6229.2} C_VEL
LIN {X 0,Y 497.471,Z 305.281,A -85,B 0,C 180,E1 -6232.422,E2 -6232.422} C_VEL
LIN {X 0,Y 497.631,Z 298.814,A -85,B 0,C 180,E1 -6233.491,E2 -6233.491} C_VEL
LIN {X 0,Y 495.823,Z 288.725,A -85,B 0,C 180,E1 -6235.277,E2 -6235.277} C_VEL
LIN {X 0,Y 495.781,Z 288.731,A -85,B 0,C 180,E1 -6237.89,E2 -6237.89} C_VEL
LIN {X 0,Y 495.749,Z 288.728,A -85,B 0,C 180,E1 -6240.686,E2 -6240.686} C_VEL
LIN {X 0,Y 495.757,Z 288.727,A -85,B 0,C 180,E1 -6243.563,E2 -6243.563} C_VEL
LIN {X 0,Y 495.729,Z 288.734,A -85,B 0,C 180,E1 -6246.543,E2 -6246.543} C_VEL
LIN {X 0,Y 495.752,Z 288.727,A -85,B 0,C 180,E1 -6249.637,E2 -6249.637} C_VEL
LIN {X 0,Y 495.733,Z 288.737,A -85,B 0,C 180,E1 -6252.506,E2 -6252.506} C_VEL
LIN {X 0,Y 495.744,Z 288.728,A -85,B 0,C 180,E1 -6255.138,E2 -6255.138} C_VEL
LIN {X 0,Y 495.772,Z 288.728,A -85,B 0,C 180,E1 -6258.22,E2 -6258.22} C_VEL
LIN {X 0,Y 495.745,Z 288.728,A -85,B 0,C 180,E1 -6261.408,E2 -6261.408} C_VEL
LIN {X 0,Y 495.748,Z 288.732,A -85,B 0,C 180,E1 -6264.462,E2 -6264.462} C_VEL
LIN {X 0,Y 495.762,Z 288.727,A -85,B 0,C 180,E1 -6267.405,E2 -6267.405} C_VEL
LIN {X 0,Y 495.773,Z 288.725,A -85,B 0,C 180,E1 -6270.254,E2 -6270.254} C_VEL
LIN {X 0,Y 495.826,Z 288.722,A -85,B 0,C 180,E1 -6273.248,E2 -6273.248} C_VEL
LIN {X 0,Y 495.744,Z 288.728,A -85,B 0,C 180,E1 -6275.724,E2 -6275.724} C_VEL
LIN {X 0,Y 495.733,Z 288.729,A -85,B 0,C 180,E1 -6278.371,E2 -6278.371} C_VEL
LIN {X 0,Y 495.775,Z 288.73,A -85,B 0,C 180,E1 -6280.971,E2 -6280.971} C_VEL
LIN {X 0,Y 495.77,Z 288.729,A -85,B 0,C 180,E1 -6283.53,E2 -6283.53} C_VEL
LIN {X 0,Y 495.789,Z 288.722,A -85,B 0,C 180,E1 -6286.056,E2 -6286.056} C_VEL
LIN {X 0,Y 495.845,Z 288.715,A -85,B 0,C 180,E1 -6288.555,E2 -6288.555} C_VEL
LIN {X 0,Y 495.864,Z 288.716,A -85,B 0,C 180,E1 -6291.852,E2 -6291.852} C_VEL
LIN {X 0,Y 495.886,Z 288.71,A -85,B 0,C 180,E1 -6294.306,E2 -6294.306} C_VEL
LIN {X 0,Y 495.982,Z 288.706,A -85,B 0,C 180,E1 -6297.564,E2 -6297.564} C_VEL
LIN {X 0,Y 495.986,Z 288.702,A -85,B 0,C 180,E1 -6300,E2 -6300} C_VEL
LIN {X 0,Y 495.983,Z 288.698,A -85,B 0,C 180,E1 -6302.436,E2 -6302.436} C_VEL
LIN {X 0,Y 495.873,Z 288.719,A -85,B 0,C 180,E1 -6305.694,E2 -6305.694} C_VEL
LIN {X 0,Y 495.832,Z 288.716,A -85,B 0,C 180,E1 -6308.97,E2 -6308.97} C_VEL
LIN {X 0,Y 495.818,Z 288.727,A -85,B 0,C 180,E1 -6312.035,E2 -6312.035} C_VEL
LIN {X 0,Y 495.814,Z 288.72,A -85,B 0,C 180,E1 -6315.452,E2 -6315.452} C_VEL
LIN {X 0,Y 495.797,Z 288.729,A -85,B 0,C 180,E1 -6318.248,E2 -6318.248} C_VEL
LIN {X 0,Y 495.765,Z 288.727,A -85,B 0,C 180,E1 -6320.757,E2 -6320.757} C_VEL
LIN {X 0,Y 495.733,Z 288.729,A -85,B 0,C 180,E1 -6323.388,E2 -6323.388} C_VEL
LIN {X 0,Y 495.796,Z 288.725,A -85,B 0,C 180,E1 -6326.746,E2 -6326.746} C_VEL
LIN {X 0,Y 495.757,Z 288.726,A -85,B 0,C 180,E1 -6329.747,E2 -6329.747} C_VEL
LIN {X 0,Y 495.759,Z 288.734,A -85,B 0,C 180,E1 -6332.595,E2 -6332.595} C_VEL
LIN {X 0,Y 495.74,Z 288.728,A -85,B 0,C 180,E1 -6335.539,E2 -6335.539} C_VEL
LIN {X 0,Y 495.751,Z 288.735,A -85,B 0,C 180,E1 -6338.768,E2 -6338.768} C_VEL
LIN {X 0,Y 495.738,Z 288.728,A -85,B 0,C 180,E1 -6341.783,E2 -6341.783} C_VEL
LIN {X 0,Y 495.731,Z 288.734,A -85,B 0,C 180,E1 -6345.142,E2 -6345.142} C_VEL
LIN {X 0,Y 495.738,Z 288.729,A -85,B 0,C 180,E1 -6348.218,E2 -6348.218} C_VEL
LIN {X 0,Y 495.741,Z 288.732,A -85,B 0,C 180,E1 -6351.409,E2 -6351.409} C_VEL
LIN {X 0,Y 495.74,Z 288.729,A -85,B 0,C 180,E1 -6354.463,E2 -6354.463} C_VEL
LIN {X 0,Y 495.761,Z 288.731,A -85,B 0,C 180,E1 -6357.406,E2 -6357.406} C_VEL
LIN {X 0,Y 495.754,Z 288.726,A -85,B 0,C 180,E1 -6360.254,E2 -6360.254} C_VEL
LIN {X 0,Y 495.722,Z 288.732,A -85,B 0,C 180,E1 -6360.74,E2 -6360.74} C_VEL
LIN {X 0,Y 495.043,Z 288.822,A -85,B 0,C 180,E1 -6361.419,E2 -6361.419} C_VEL
LIN {X 0,Y 492.167,Z 289.179,A -85,B 0,C 180,E1 -6362.521,E2 -6362.521} C_VEL
LIN {X 0,Y 489.75,Z 289.483,A -85,B 0,C 180,E1 -6363.409,E2 -6363.409} C_VEL
LIN {X 0,Y 488.727,Z 289.603,A -85,B 0,C 180,E1 -6364.095,E2 -6364.095} C_VEL
LIN {X 0,Y 488.652,Z 289.611,A -85,B 0,C 180,E1 -6364.327,E2 -6364.327} C_VEL
LIN {X 0,Y 488.72,Z 289.607,A -85,B 0,C 180,E1 -6367.154,E2 -6367.154} C_VEL
LIN {X 0,Y 488.723,Z 289.607,A -85,B 0,C 180,E1 -6369.811,E2 -6369.811} C_VEL
LIN {X 0,Y 488.7,Z 289.605,A -85,B 0,C 180,E1 -6372.423,E2 -6372.423} C_VEL
LIN {X 0,Y 488.755,Z 289.599,A -85,B 0,C 180,E1 -6375,E2 -6375} C_VEL
LIN {X 0,Y 488.759,Z 289.599,A -85,B 0,C 180,E1 -6378.387,E2 -6378.387} C_VEL
LIN {X 0,Y 488.754,Z 289.608,A -85,B 0,C 180,E1 -6381.733,E2 -6381.733} C_VEL
LIN {X 0,Y 488.837,Z 289.738,A -85,B 0,C 180,E1 -6383.759,E2 -6383.759} C_VEL
LIN {X 0,Y 489.476,Z 295.128,A -85,B 0,C 180,E1 -6384.852,E2 -6384.852} C_VEL
LIN {X 0,Y 489.292,Z 308.862,A -85,B 0,C 180,E1 -6387.531,E2 -6387.531} C_VEL
LIN {X 0,Y 489.238,Z 310.343,A -85,B 0,C 180,E1 -6387.802,E2 -6387.802} C_VEL
LIN {X 0,Y 491.766,Z 323.514,A -85,B 0,C 180,E1 -6388.083,E2 -6388.083} C_VEL
LIN {X 0,Y 491.183,Z 417.564,A -85,B 0,C 180,E1 -6389.488,E2 -6389.488} C_VEL
LIN {X 0,Y 490.88,Z 429.885,A -85,B 0,C 180,E1 -6389.821,E2 -6389.821} C_VEL
LIN {X 0,Y 490.611,Z 443.121,A -85,B 0,C 180,E1 -6390.36,E2 -6390.36} C_VEL
LIN {X 0,Y 490.228,Z 455.1,A -85,B 0,C 180,E1 -6391.027,E2 -6391.027} C_VEL
LIN {X 0,Y 489.806,Z 466.501,A -85,B 0,C 180,E1 -6391.851,E2 -6391.851} C_VEL
LIN {X 0,Y 489.39,Z 476.791,A -85,B 0,C 180,E1 -6392.779,E2 -6392.779} C_VEL
LIN {X 0,Y 489.026,Z 485.227,A -85,B 0,C 180,E1 -6393.709,E2 -6393.709} C_VEL
LIN {X 0,Y 488.753,Z 493.008,A -85,B 0,C 180,E1 -6394.743,E2 -6394.743} C_VEL
LIN {X 0,Y 488.453,Z 500.638,A -85,B 0,C 180,E1 -6395.988,E2 -6395.988} C_VEL
LIN {X 0,Y 488.249,Z 507.676,A -85,B 0,C 180,E1 -6397.444,E2 -6397.444} C_VEL
LIN {X 0,Y 488.074,Z 512.377,A -85,B 0,C 180,E1 -6398.697,E2 -6398.697} C_VEL
LIN {X 0,Y 487.993,Z 515.967,A -85,B 0,C 180,E1 -6399.952,E2 -6399.952} C_VEL
LIN {X 0,Y 487.946,Z 517.808,A -85,B 0,C 180,E1 -6400.792,E2 -6400.792} C_VEL
LIN {X 0,Y 487.931,Z 519.183,A -85,B 0,C 180,E1 -6401.634,E2 -6401.634} C_VEL
LIN {X 0,Y 487.837,Z 520.744,A -85,B 0,C 180,E1 -6403.327,E2 -6403.327} C_VEL
LIN {X 0,Y 487.837,Z 520.88,A -85,B 0,C 180,E1 -6404.177,E2 -6404.177} C_VEL
LIN {X 0,Y 487.863,Z 520.52,A -85,B 0,C 180,E1 -6405.163,E2 -6405.163} C_VEL
LIN {X 0,Y 487.829,Z 518.795,A -85,B 0,C 180,E1 -6406.747,E2 -6406.747} C_VEL
LIN {X 0,Y 487.979,Z 516.115,A -85,B 0,C 180,E1 -6408.093,E2 -6408.093} C_VEL
LIN {X 0,Y 488.086,Z 512.607,A -85,B 0,C 180,E1 -6409.341,E2 -6409.341} C_VEL
LIN {X 0,Y 488.275,Z 507.606,A -85,B 0,C 180,E1 -6410.677,E2 -6410.677} C_VEL
LIN {X 0,Y 488.425,Z 501.433,A -85,B 0,C 180,E1 -6411.97,E2 -6411.97} C_VEL
LIN {X 0,Y 488.802,Z 493.272,A -85,B 0,C 180,E1 -6413.325,E2 -6413.325} C_VEL
LIN {X 0,Y 489.087,Z 485.198,A -85,B 0,C 180,E1 -6414.402,E2 -6414.402} C_VEL
LIN {X 0,Y 489.487,Z 474.903,A -85,B 0,C 180,E1 -6415.515,E2 -6415.515} C_VEL
LIN {X 0,Y 489.882,Z 464.676,A -85,B 0,C 180,E1 -6416.407,E2 -6416.407} C_VEL
LIN {X 0,Y 490.388,Z 453.008,A -85,B 0,C 180,E1 -6417.21,E2 -6417.21} C_VEL
LIN {X 0,Y 490.649,Z 440.767,A -85,B 0,C 180,E1 -6417.86,E2 -6417.86} C_VEL
LIN {X 0,Y 490.938,Z 428.472,A -85,B 0,C 180,E1 -6418.337,E2 -6418.337} C_VEL
LIN {X 0,Y 491.143,Z 414.921,A -85,B 0,C 180,E1 -6418.674,E2 -6418.674} C_VEL
LIN {X 0,Y 491.726,Z 322.607,A -85,B 0,C 180,E1 -6420.047,E2 -6420.047} C_VEL
LIN {X 0,Y 489.33,Z 310.088,A -85,B 0,C 180,E1 -6420.338,E2 -6420.338} C_VEL
LIN {X 0,Y 489.547,Z 295.615,A -85,B 0,C 180,E1 -6423.061,E2 -6423.061} C_VEL
LIN {X 0,Y 488.889,Z 290.313,A -85,B 0,C 180,E1 -6424.1,E2 -6424.1} C_VEL
LIN {X 0,Y 488.727,Z 289.611,A -85,B 0,C 180,E1 -6424.3,E2 -6424.3} C_VEL
LIN {X 0,Y 488.68,Z 289.61,A -85,B 0,C 180,E1 -6427.722,E2 -6427.722} C_VEL
LIN {X 0,Y 488.721,Z 289.611,A -85,B 0,C 180,E1 -6430.345,E2 -6430.345} C_VEL
LIN {X 0,Y 488.686,Z 289.61,A -85,B 0,C 180,E1 -6433.655,E2 -6433.655} C_VEL
LIN {X 0,Y 488.686,Z 289.613,A -85,B 0,C 180,E1 -6436.345,E2 -6436.345} C_VEL
LIN {X 0,Y 488.735,Z 289.602,A -85,B 0,C 180,E1 -6439.676,E2 -6439.676} C_VEL
LIN {X 0,Y 488.68,Z 289.617,A -85,B 0,C 180,E1 -6442.841,E2 -6442.841} C_VEL
LIN {X 0,Y 488.731,Z 289.602,A -85,B 0,C 180,E1 -6445.887,E2 -6445.887} C_VEL
LIN {X 0,Y 488.693,Z 289.614,A -85,B 0,C 180,E1 -6448.82,E2 -6448.82} C_VEL
LIN {X 0,Y 488.745,Z 289.601,A -85,B 0,C 180,E1 -6451.671,E2 -6451.671} C_VEL
LIN {X 0,Y 488.748,Z 289.6,A -85,B 0,C 180,E1 -6454.444,E2 -6454.444} C_VEL
LIN {X 0,Y 488.723,Z 289.607,A -85,B 0,C 180,E1 -6457.153,E2 -6457.153} C_VEL
LIN {X 0,Y 488.725,Z 289.603,A -85,B 0,C 180,E1 -6459.81,E2 -6459.81} C_VEL
LIN {X 0,Y 488.729,Z 289.601,A -85,B 0,C 180,E1 -6462.423,E2 -6462.423} C_VEL
LIN {X 0,Y 488.762,Z 289.599,A -85,B 0,C 180,E1 -6465,E2 -6465} C_VEL
LIN {X 0,Y 488.805,Z 289.592,A -85,B 0,C 180,E1 -6468.387,E2 -6468.387} C_VEL
LIN {X 0,Y 488.817,Z 289.596,A -85,B 0,C 180,E1 -6471.734,E2 -6471.734} C_VEL
LIN {X 0,Y 488.846,Z 289.588,A -85,B 0,C 180,E1 -6474.224,E2 -6474.224} C_VEL
LIN {X 0,Y 488.96,Z 289.575,A -85,B 0,C 180,E1 -6477.529,E2 -6477.529} C_VEL
LIN {X 0,Y 488.933,Z 289.57,A -85,B 0,C 180,E1 -6480.824,E2 -6480.824} C_VEL
LIN {X 0,Y 488.96,Z 289.575,A -85,B 0,C 180,E1 -6482.471,E2 -6482.471} C_VEL
LIN {X 0,Y 488.846,Z 289.588,A -85,B 0,C 180,E1 -6485.776,E2 -6485.776} C_VEL
LIN {X 0,Y 488.816,Z 289.598,A -85,B 0,C 180,E1 -6488.266,E2 -6488.266} C_VEL
LIN {X 0,Y 488.805,Z 289.587,A -85,B 0,C 180,E1 -6491.612,E2 -6491.612} C_VEL
LIN {X 0,Y 488.762,Z 289.597,A -85,B 0,C 180,E1 -6495,E2 -6495} C_VEL
LIN {X 0,Y 488.755,Z 289.605,A -85,B 0,C 180,E1 -6498.442,E2 -6498.442} C_VEL
LIN {X 0,Y 488.707,Z 289.605,A -85,B 0,C 180,E1 -6501.071,E2 -6501.071} C_VEL
LIN {X 0,Y 488.689,Z 289.607,A -85,B 0,C 180,E1 -6503.746,E2 -6503.746} C_VEL
LIN {X 0,Y 488.792,Z 289.602,A -85,B 0,C 180,E1 -6506.944,E2 -6506.944} C_VEL
LIN {X 0,Y 488.71,Z 289.602,A -85,B 0,C 180,E1 -6510.363,E2 -6510.363} C_VEL
LIN {X 0,Y 488.729,Z 289.602,A -85,B 0,C 180,E1 -6513.483,E2 -6513.483} C_VEL
LIN {X 0,Y 488.683,Z 289.608,A -85,B 0,C 180,E1 -6516.355,E2 -6516.355} C_VEL
LIN {X 0,Y 488.702,Z 289.613,A -85,B 0,C 180,E1 -6519.254,E2 -6519.254} C_VEL
LIN {X 0,Y 488.708,Z 289.61,A -85,B 0,C 180,E1 -6521.6,E2 -6521.6} C_VEL
LIN {X 0,Y 488.702,Z 289.608,A -85,B 0,C 180,E1 -6524.803,E2 -6524.803} C_VEL
LIN {X 0,Y 488.693,Z 289.614,A -85,B 0,C 180,E1 -6527.475,E2 -6527.475} C_VEL
LIN {X 0,Y 488.735,Z 289.606,A -85,B 0,C 180,E1 -6529.677,E2 -6529.677} C_VEL
LIN {X 0,Y 488.681,Z 289.61,A -85,B 0,C 180,E1 -6532.841,E2 -6532.841} C_VEL
LIN {X 0,Y 488.732,Z 289.608,A -85,B 0,C 180,E1 -6535.887,E2 -6535.887} C_VEL
LIN {X 0,Y 488.694,Z 289.606,A -85,B 0,C 180,E1 -6538.82,E2 -6538.82} C_VEL
LIN {X 0,Y 488.746,Z 289.607,A -85,B 0,C 180,E1 -6541.671,E2 -6541.671} C_VEL
LIN {X 0,Y 488.793,Z 289.724,A -85,B 0,C 180,E1 -6544.545,E2 -6544.545} C_VEL
LIN {X 0,Y 490.694,Z 300.21,A -85,B 0,C 180,E1 -6546.441,E2 -6546.441} C_VEL
LIN {X 0,Y 490.243,Z 313.819,A -85,B 0,C 180,E1 -6548.721,E2 -6548.721} C_VEL
LIN {X 0,Y 489.583,Z 333.85,A -85,B 0,C 180,E1 -6552.023,E2 -6552.023} C_VEL
LIN {X 0,Y 489.252,Z 344.235,A -85,B 0,C 180,E1 -6553.713,E2 -6553.713} C_VEL
LIN {X 0,Y 491.666,Z 360.627,A -85,B 0,C 180,E1 -6554.044,E2 -6554.044} C_VEL
LIN {X 0,Y 491.096,Z 452.605,A -85,B 0,C 180,E1 -6555.417,E2 -6555.417} C_VEL
LIN {X 0,Y 490.761,Z 465.892,A -85,B 0,C 180,E1 -6555.777,E2 -6555.777} C_VEL
LIN {X 0,Y 490.424,Z 478.072,A -85,B 0,C 180,E1 -6556.269,E2 -6556.269} C_VEL
LIN {X 0,Y 489.975,Z 490.627,A -85,B 0,C 180,E1 -6556.96,E2 -6556.96} C_VEL
LIN {X 0,Y 489.583,Z 501.991,A -85,B 0,C 180,E1 -6557.775,E2 -6557.775} C_VEL
LIN {X 0,Y 489.2,Z 512.458,A -85,B 0,C 180,E1 -6558.712,E2 -6558.712} C_VEL
LIN {X 0,Y 488.836,Z 521.018,A -85,B 0,C 180,E1 -6559.647,E2 -6559.647} C_VEL
LIN {X 0,Y 488.521,Z 528.921,A -85,B 0,C 180,E1 -6560.685,E2 -6560.685} C_VEL
LIN {X 0,Y 488.276,Z 536.644,A -85,B 0,C 180,E1 -6561.932,E2 -6561.932} C_VEL
LIN {X 0,Y 488.074,Z 543.764,A -85,B 0,C 180,E1 -6563.385,E2 -6563.385} C_VEL
LIN {X 0,Y 488.018,Z 548.508,A -85,B 0,C 180,E1 -6564.628,E2 -6564.628} C_VEL
LIN {X 0,Y 487.929,Z 552.133,A -85,B 0,C 180,E1 -6565.87,E2 -6565.87} C_VEL
LIN {X 0,Y 487.964,Z 554.006,A -85,B 0,C 180,E1 -6566.697,E2 -6566.697} C_VEL
LIN {X 0,Y 487.89,Z 556.411,A -85,B 0,C 180,E1 -6568.349,E2 -6568.349} C_VEL
LIN {X 0,Y 487.822,Z 557.242,A -85,B 0,C 180,E1 -6569.999,E2 -6569.999} C_VEL
LIN {X 0,Y 487.89,Z 556.424,A -85,B 0,C 180,E1 -6571.65,E2 -6571.65} C_VEL
LIN {X 0,Y 487.908,Z 555.429,A -85,B 0,C 180,E1 -6572.476,E2 -6572.476} C_VEL
LIN {X 0,Y 487.964,Z 554.033,A -85,B 0,C 180,E1 -6573.302,E2 -6573.302} C_VEL
LIN {X 0,Y 487.92,Z 551.09,A -85,B 0,C 180,E1 -6574.543,E2 -6574.543} C_VEL
LIN {X 0,Y 488.021,Z 547.109,A -85,B 0,C 180,E1 -6575.785,E2 -6575.785} C_VEL
LIN {X 0,Y 488.179,Z 540.984,A -85,B 0,C 180,E1 -6577.236,E2 -6577.236} C_VEL
LIN {X 0,Y 488.356,Z 534.286,A -85,B 0,C 180,E1 -6578.482,E2 -6578.482} C_VEL
LIN {X 0,Y 488.646,Z 525.976,A -85,B 0,C 180,E1 -6579.729,E2 -6579.729} C_VEL
LIN {X 0,Y 488.991,Z 517.454,A -85,B 0,C 180,E1 -6580.768,E2 -6580.768} C_VEL
LIN {X 0,Y 489.438,Z 506.925,A -85,B 0,C 180,E1 -6581.806,E2 -6581.806} C_VEL
LIN {X 0,Y 489.81,Z 495.54,A -85,B 0,C 180,E1 -6582.709,E2 -6582.709} C_VEL
LIN {X 0,Y 490.228,Z 483.12,A -85,B 0,C 180,E1 -6583.471,E2 -6583.471} C_VEL
LIN {X 0,Y 490.665,Z 470.691,A -85,B 0,C 180,E1 -6584.039,E2 -6584.039} C_VEL
LIN {X 0,Y 490.92,Z 457.862,A -85,B 0,C 180,E1 -6584.455,E2 -6584.455} C_VEL
LIN {X 0,Y 491.167,Z 444.26,A -85,B 0,C 180,E1 -6584.712,E2 -6584.712} C_VEL
LIN {X 0,Y 491.581,Z 359.613,A -85,B 0,C 180,E1 -6585.959,E2 -6585.959} C_VEL
LIN {X 0,Y 489.258,Z 344.374,A -85,B 0,C 180,E1 -6586.266,E2 -6586.266} C_VEL
LIN {X 0,Y 489.891,Z 324.697,A -85,B 0,C 180,E1 -6589.483,E2 -6589.483} C_VEL
LIN {X 0,Y 490.554,Z 304.943,A -85,B 0,C 180,E1 -6592.756,E2 -6592.756} C_VEL
LIN {X 0,Y 490.646,Z 299.66,A -85,B 0,C 180,E1 -6593.644,E2 -6593.644} C_VEL
LIN {X 0,Y 488.793,Z 289.602,A -85,B 0,C 180,E1 -6595.454,E2 -6595.454} C_VEL
LIN {X 0,Y 488.743,Z 289.608,A -85,B 0,C 180,E1 -6598.328,E2 -6598.328} C_VEL
LIN {X 0,Y 488.689,Z 289.606,A -85,B 0,C 180,E1 -6601.179,E2 -6601.179} C_VEL
LIN {X 0,Y 488.731,Z 289.609,A -85,B 0,C 180,E1 -6604.112,E2 -6604.112} C_VEL
LIN {X 0,Y 488.678,Z 289.608,A -85,B 0,C 180,E1 -6607.158,E2 -6607.158} C_VEL
LIN {X 0,Y 488.713,Z 289.613,A -85,B 0,C 180,E1 -6610.344,E2 -6610.344} C_VEL
LIN {X 0,Y 488.682,Z 289.607,A -85,B 0,C 180,E1 -6613.653,E2 -6613.653} C_VEL
LIN {X 0,Y 488.687,Z 289.613,A -85,B 0,C 180,E1 -6616.345,E2 -6616.345} C_VEL
LIN {X 0,Y 488.714,Z 289.613,A -85,B 0,C 180,E1 -6618.585,E2 -6618.585} C_VEL
LIN {X 0,Y 488.675,Z 289.608,A -85,B 0,C 180,E1 -6621.799,E2 -6621.799} C_VEL
LIN {X 0,Y 488.72,Z 289.607,A -85,B 0,C 180,E1 -6625.051,E2 -6625.051} C_VEL
LIN {X 0,Y 488.699,Z 289.605,A -85,B 0,C 180,E1 -6628.045,E2 -6628.045} C_VEL
LIN {X 0,Y 488.725,Z 289.608,A -85,B 0,C 180,E1 -6630.73,E2 -6630.73} C_VEL
LIN {X 0,Y 488.758,Z 289.599,A -85,B 0,C 180,E1 -6633.528,E2 -6633.528} C_VEL
LIN {X 0,Y 488.684,Z 289.607,A -85,B 0,C 180,E1 -6636.254,E2 -6636.254} C_VEL
LIN {X 0,Y 488.737,Z 289.609,A -85,B 0,C 180,E1 -6639.175,E2 -6639.175} C_VEL
LIN {X 0,Y 488.724,Z 289.602,A -85,B 0,C 180,E1 -6642.423,E2 -6642.423} C_VEL
LIN {X 0,Y 488.755,Z 289.603,A -85,B 0,C 180,E1 -6644.999,E2 -6644.999} C_VEL
LIN {X 0,Y 488.798,Z 289.592,A -85,B 0,C 180,E1 -6648.387,E2 -6648.387} C_VEL
LIN {X 0,Y 488.809,Z 289.596,A -85,B 0,C 180,E1 -6651.733,E2 -6651.733} C_VEL
LIN {X 0,Y 488.845,Z 289.587,A -85,B 0,C 180,E1 -6654.224,E2 -6654.224} C_VEL
LIN {X 0,Y 488.95,Z 289.582,A -85,B 0,C 180,E1 -6657.529,E2 -6657.529} C_VEL
LIN {X 0,Y 488.944,Z 289.574,A -85,B 0,C 180,E1 -6660.824,E2 -6660.824} C_VEL
LIN {X 0,Y 488.951,Z 289.574,A -85,B 0,C 180,E1 -6662.471,E2 -6662.471} C_VEL
LIN {X 0,Y 488.83,Z 289.597,A -85,B 0,C 180,E1 -6665.776,E2 -6665.776} C_VEL
LIN {X 0,Y 488.807,Z 289.595,A -85,B 0,C 180,E1 -6668.267,E2 -6668.267} C_VEL
LIN {X 0,Y 488.795,Z 289.597,A -85,B 0,C 180,E1 -6671.613,E2 -6671.613} C_VEL
LIN {X 0,Y 488.751,Z 289.598,A -85,B 0,C 180,E1 -6675.001,E2 -6675.001} C_VEL
LIN {X 0,Y 488.746,Z 289.604,A -85,B 0,C 180,E1 -6678.443,E2 -6678.443} C_VEL
LIN {X 0,Y 488.697,Z 289.605,A -85,B 0,C 180,E1 -6681.071,E2 -6681.071} C_VEL
LIN {X 0,Y 488.666,Z 289.611,A -85,B 0,C 180,E1 -6683.747,E2 -6683.747} C_VEL
LIN {X 0,Y 488.737,Z 289.602,A -85,B 0,C 180,E1 -6686.934,E2 -6686.934} C_VEL
LIN {X 0,Y 488.715,Z 289.608,A -85,B 0,C 180,E1 -6690.22,E2 -6690.22} C_VEL
LIN {X 0,Y 488.727,Z 289.601,A -85,B 0,C 180,E1 -6693.485,E2 -6693.485} C_VEL
LIN {X 0,Y 488.675,Z 289.613,A -85,B 0,C 180,E1 -6696.355,E2 -6696.355} C_VEL
LIN {X 0,Y 488.687,Z 289.608,A -85,B 0,C 180,E1 -6699.256,E2 -6699.256} C_VEL
LIN {X 0,Y 488.681,Z 289.612,A -85,B 0,C 180,E1 -6702.527,E2 -6702.527} C_VEL
LIN {X 0,Y 488.695,Z 289.61,A -85,B 0,C 180,E1 -6705.198,E2 -6705.198} C_VEL
LIN {X 0,Y 488.671,Z 289.612,A -85,B 0,C 180,E1 -6708.582,E2 -6708.582} C_VEL
LIN {X 0,Y 488.693,Z 289.614,A -85,B 0,C 180,E1 -6710.949,E2 -6710.949} C_VEL
LIN {X 0,Y 488.666,Z 289.61,A -85,B 0,C 180,E1 -6713.868,E2 -6713.868} C_VEL
LIN {X 0,Y 488.732,Z 289.605,A -85,B 0,C 180,E1 -6716.878,E2 -6716.878} C_VEL
LIN {X 0,Y 488.713,Z 289.605,A -85,B 0,C 180,E1 -6719.781,E2 -6719.781} C_VEL
LIN {X 0,Y 488.694,Z 289.611,A -85,B 0,C 180,E1 -6723.08,E2 -6723.08} C_VEL
LIN {X 0,Y 488.652,Z 289.611,A -85,B 0,C 180,E1 -6724.327,E2 -6724.327} C_VEL
LIN {X 0,Y 488.009,Z 289.696,A -85,B 0,C 180,E1 -6725.016,E2 -6725.016} C_VEL
LIN {X 0,Y 485.177,Z 290.05,A -85,B 0,C 180,E1 -6726.133,E2 -6726.133} C_VEL
LIN {X 0,Y 482.765,Z 290.352,A -85,B 0,C 180,E1 -6727.034,E2 -6727.034} C_VEL
LIN {X 0,Y 481.723,Z 290.48,A -85,B 0,C 180,E1 -6727.73,E2 -6727.73} C_VEL
LIN {X 0,Y 481.635,Z 290.487,A -85,B 0,C 180,E1 -6727.966,E2 -6727.966} C_VEL
LIN {X 0,Y 481.7,Z 290.477,A -85,B 0,C 180,E1 -6730.394,E2 -6730.394} C_VEL
LIN {X 0,Y 481.665,Z 290.483,A -85,B 0,C 180,E1 -6733.034,E2 -6733.034} C_VEL
LIN {X 0,Y 481.673,Z 290.489,A -85,B 0,C 180,E1 -6735.639,E2 -6735.639} C_VEL
LIN {X 0,Y 481.714,Z 290.478,A -85,B 0,C 180,E1 -6738.215,E2 -6738.215} C_VEL
LIN {X 0,Y 481.712,Z 290.484,A -85,B 0,C 180,E1 -6741.612,E2 -6741.612} C_VEL
LIN {X 0,Y 481.789,Z 290.586,A -85,B 0,C 180,E1 -6743.615,E2 -6743.615} C_VEL
LIN {X 0,Y 482.495,Z 296.271,A -85,B 0,C 180,E1 -6744.777,E2 -6744.777} C_VEL
LIN {X 0,Y 482.337,Z 307.949,A -85,B 0,C 180,E1 -6747.077,E2 -6747.077} C_VEL
LIN {X 0,Y 482.254,Z 310.539,A -85,B 0,C 180,E1 -6747.573,E2 -6747.573} C_VEL
LIN {X 0,Y 484.944,Z 324.298,A -85,B 0,C 180,E1 -6747.872,E2 -6747.872} C_VEL
LIN {X 0,Y 484.31,Z 417.221,A -85,B 0,C 180,E1 -6749.273,E2 -6749.273} C_VEL
LIN {X 0,Y 484.015,Z 429.742,A -85,B 0,C 180,E1 -6749.611,E2 -6749.611} C_VEL
LIN {X 0,Y 483.716,Z 443.107,A -85,B 0,C 180,E1 -6750.157,E2 -6750.157} C_VEL
LIN {X 0,Y 483.318,Z 455.179,A -85,B 0,C 180,E1 -6750.834,E2 -6750.834} C_VEL
LIN {X 0,Y 482.862,Z 466.632,A -85,B 0,C 180,E1 -6751.669,E2 -6751.669} C_VEL
LIN {X 0,Y 482.419,Z 476.957,A -85,B 0,C 180,E1 -6752.61,E2 -6752.61} C_VEL
LIN {X 0,Y 482.024,Z 485.411,A -85,B 0,C 180,E1 -6753.553,E2 -6753.553} C_VEL
LIN {X 0,Y 481.723,Z 493.209,A -85,B 0,C 180,E1 -6754.603,E2 -6754.603} C_VEL
LIN {X 0,Y 481.403,Z 500.853,A -85,B 0,C 180,E1 -6755.866,E2 -6755.866} C_VEL
LIN {X 0,Y 481.245,Z 506.81,A -85,B 0,C 180,E1 -6757.089,E2 -6757.089} C_VEL
LIN {X 0,Y 481.038,Z 511.891,A -85,B 0,C 180,E1 -6758.402,E2 -6758.402} C_VEL
LIN {X 0,Y 480.924,Z 515.67,A -85,B 0,C 180,E1 -6759.675,E2 -6759.675} C_VEL
LIN {X 0,Y 480.851,Z 518.423,A -85,B 0,C 180,E1 -6760.954,E2 -6760.954} C_VEL
LIN {X 0,Y 480.813,Z 519.721,A -85,B 0,C 180,E1 -6761.809,E2 -6761.809} C_VEL
LIN {X 0,Y 480.762,Z 520.62,A -85,B 0,C 180,E1 -6762.667,E2 -6762.667} C_VEL
LIN {X 0,Y 480.734,Z 521.068,A -85,B 0,C 180,E1 -6763.528,E2 -6763.528} C_VEL
LIN {X 0,Y 480.75,Z 521.106,A -85,B 0,C 180,E1 -6764.39,E2 -6764.39} C_VEL
LIN {X 0,Y 480.757,Z 520.744,A -85,B 0,C 180,E1 -6765.257,E2 -6765.257} C_VEL
LIN {X 0,Y 480.712,Z 519.958,A -85,B 0,C 180,E1 -6766.128,E2 -6766.128} C_VEL
LIN {X 0,Y 480.754,Z 518.701,A -85,B 0,C 180,E1 -6767.001,E2 -6767.001} C_VEL
LIN {X 0,Y 480.917,Z 516.238,A -85,B 0,C 180,E1 -6768.214,E2 -6768.214} C_VEL
LIN {X 0,Y 481.033,Z 512.158,A -85,B 0,C 180,E1 -6769.636,E2 -6769.636} C_VEL
LIN {X 0,Y 481.232,Z 506.788,A -85,B 0,C 180,E1 -6771.034,E2 -6771.034} C_VEL
LIN {X 0,Y 481.449,Z 500.569,A -85,B 0,C 180,E1 -6772.305,E2 -6772.305} C_VEL
LIN {X 0,Y 481.776,Z 493.818,A -85,B 0,C 180,E1 -6773.423,E2 -6773.423} C_VEL
LIN {X 0,Y 482.097,Z 485.549,A -85,B 0,C 180,E1 -6774.549,E2 -6774.549} C_VEL
LIN {X 0,Y 482.478,Z 476.298,A -85,B 0,C 180,E1 -6775.578,E2 -6775.578} C_VEL
LIN {X 0,Y 482.956,Z 465.108,A -85,B 0,C 180,E1 -6776.582,E2 -6776.582} C_VEL
LIN {X 0,Y 483.43,Z 454.828,A -85,B 0,C 180,E1 -6777.316,E2 -6777.316} C_VEL
LIN {X 0,Y 483.759,Z 442.595,A -85,B 0,C 180,E1 -6777.998,E2 -6777.998} C_VEL
LIN {X 0,Y 484.062,Z 429.635,A -85,B 0,C 180,E1 -6778.525,E2 -6778.525} C_VEL
LIN {X 0,Y 484.298,Z 417.658,A -85,B 0,C 180,E1 -6778.85,E2 -6778.85} C_VEL
LIN {X 0,Y 485.053,Z 324.086,A -85,B 0,C 180,E1 -6780.267,E2 -6780.267} C_VEL
LIN {X 0,Y 482.35,Z 310.282,A -85,B 0,C 180,E1 -6780.602,E2 -6780.602} C_VEL
LIN {X 0,Y 482.604,Z 297.168,A -85,B 0,C 180,E1 -6783.1,E2 -6783.1} C_VEL
LIN {X 0,Y 482.259,Z 293.418,A -85,B 0,C 180,E1 -6783.832,E2 -6783.832} C_VEL
LIN {X 0,Y 481.718,Z 290.484,A -85,B 0,C 180,E1 -6784.451,E2 -6784.451} C_VEL
LIN {X 0,Y 481.657,Z 290.489,A -85,B 0,C 180,E1 -6788.007,E2 -6788.007} C_VEL
LIN {X 0,Y 481.658,Z 290.486,A -85,B 0,C 180,E1 -6791.042,E2 -6791.042} C_VEL
LIN {X 0,Y 481.657,Z 290.492,A -85,B 0,C 180,E1 -6794.458,E2 -6794.458} C_VEL
LIN {X 0,Y 481.649,Z 290.486,A -85,B 0,C 180,E1 -6797.839,E2 -6797.839} C_VEL
LIN {X 0,Y 481.681,Z 290.482,A -85,B 0,C 180,E1 -6800.651,E2 -6800.651} C_VEL
LIN {X 0,Y 481.628,Z 290.489,A -85,B 0,C 180,E1 -6803.376,E2 -6803.376} C_VEL
LIN {X 0,Y 481.711,Z 290.479,A -85,B 0,C 180,E1 -6806.33,E2 -6806.33} C_VEL
LIN {X 0,Y 481.651,Z 290.484,A -85,B 0,C 180,E1 -6809.417,E2 -6809.417} C_VEL
LIN {X 0,Y 481.7,Z 290.478,A -85,B 0,C 180,E1 -6812.168,E2 -6812.168} C_VEL
LIN {X 0,Y 481.718,Z 290.481,A -85,B 0,C 180,E1 -6814.97,E2 -6814.97} C_VEL
LIN {X 0,Y 481.649,Z 290.486,A -85,B 0,C 180,E1 -6817.705,E2 -6817.705} C_VEL
LIN {X 0,Y 481.705,Z 290.475,A -85,B 0,C 180,E1 -6820.393,E2 -6820.393} C_VEL
LIN {X 0,Y 481.688,Z 290.481,A -85,B 0,C 180,E1 -6823.034,E2 -6823.034} C_VEL
LIN {X 0,Y 481.69,Z 290.482,A -85,B 0,C 180,E1 -6825.639,E2 -6825.639} C_VEL
LIN {X 0,Y 481.75,Z 290.472,A -85,B 0,C 180,E1 -6828.215,E2 -6828.215} C_VEL
LIN {X 0,Y 481.762,Z 290.472,A -85,B 0,C 180,E1 -6831.612,E2 -6831.612} C_VEL
LIN {X 0,Y 481.807,Z 290.466,A -85,B 0,C 180,E1 -6834.139,E2 -6834.139} C_VEL
LIN {X 0,Y 481.927,Z 290.45,A -85,B 0,C 180,E1 -6837.492,E2 -6837.492} C_VEL
LIN {X 0,Y 481.885,Z 290.448,A -85,B 0,C 180,E1 -6840.836,E2 -6840.836} C_VEL
LIN {X 0,Y 481.927,Z 290.451,A -85,B 0,C 180,E1 -6842.507,E2 -6842.507} C_VEL
LIN {X 0,Y 481.806,Z 290.466,A -85,B 0,C 180,E1 -6845.861,E2 -6845.861} C_VEL
LIN {X 0,Y 481.761,Z 290.475,A -85,B 0,C 180,E1 -6848.388,E2 -6848.388} C_VEL
LIN {X 0,Y 481.75,Z 290.466,A -85,B 0,C 180,E1 -6851.785,E2 -6851.785} C_VEL
LIN {X 0,Y 481.742,Z 290.47,A -85,B 0,C 180,E1 -6855.224,E2 -6855.224} C_VEL
LIN {X 0,Y 481.712,Z 290.482,A -85,B 0,C 180,E1 -6858.722,E2 -6858.722} C_VEL
LIN {X 0,Y 481.645,Z 290.482,A -85,B 0,C 180,E1 -6861.395,E2 -6861.395} C_VEL
LIN {X 0,Y 481.674,Z 290.482,A -85,B 0,C 180,E1 -6864.113,E2 -6864.113} C_VEL
LIN {X 0,Y 481.747,Z 290.476,A -85,B 0,C 180,E1 -6867.139,E2 -6867.139} C_VEL
LIN {X 0,Y 481.679,Z 290.476,A -85,B 0,C 180,E1 -6869.741,E2 -6869.741} C_VEL
LIN {X 0,Y 481.67,Z 290.485,A -85,B 0,C 180,E1 -6872.674,E2 -6872.674} C_VEL
LIN {X 0,Y 481.636,Z 290.487,A -85,B 0,C 180,E1 -6875.71,E2 -6875.71} C_VEL
LIN {X 0,Y 481.672,Z 290.485,A -85,B 0,C 180,E1 -6878.859,E2 -6878.859} C_VEL
LIN {X 0,Y 481.654,Z 290.486,A -85,B 0,C 180,E1 -6881.913,E2 -6881.913} C_VEL
LIN {X 0,Y 481.656,Z 290.484,A -85,B 0,C 180,E1 -6884.458,E2 -6884.458} C_VEL
LIN {X 0,Y 481.649,Z 290.489,A -85,B 0,C 180,E1 -6887.839,E2 -6887.839} C_VEL
LIN {X 0,Y 481.663,Z 290.479,A -85,B 0,C 180,E1 -6890.654,E2 -6890.654} C_VEL
LIN {X 0,Y 481.629,Z 290.493,A -85,B 0,C 180,E1 -6893.376,E2 -6893.376} C_VEL
LIN {X 0,Y 481.712,Z 290.477,A -85,B 0,C 180,E1 -6896.33,E2 -6896.33} C_VEL
LIN {X 0,Y 481.653,Z 290.486,A -85,B 0,C 180,E1 -6899.417,E2 -6899.417} C_VEL
LIN {X 0,Y 481.702,Z 290.484,A -85,B 0,C 180,E1 -6902.168,E2 -6902.168} C_VEL
LIN {X 0,Y 481.77,Z 290.599,A -85,B 0,C 180,E1 -6904.324,E2 -6904.324} C_VEL
LIN {X 0,Y 483.696,Z 301.093,A -85,B 0,C 180,E1 -6906.26,E2 -6906.26} C_VEL
LIN {X 0,Y 483.427,Z 311.488,A -85,B 0,C 180,E1 -6908.035,E2 -6908.035} C_VEL
LIN {X 0,Y 482.728,Z 331.03,A -85,B 0,C 180,E1 -6911.319,E2 -6911.319} C_VEL
LIN {X 0,Y 482.274,Z 344.006,A -85,B 0,C 180,E1 -6913.459,E2 -6913.459} C_VEL
LIN {X 0,Y 484.864,Z 361.119,A -85,B 0,C 180,E1 -6913.814,E2 -6913.814} C_VEL
LIN {X 0,Y 484.245,Z 452.712,A -85,B 0,C 180,E1 -6915.206,E2 -6915.206} C_VEL
LIN {X 0,Y 483.893,Z 465.851,A -85,B 0,C 180,E1 -6915.571,E2 -6915.571} C_VEL
LIN {X 0,Y 483.526,Z 477.95,A -85,B 0,C 180,E1 -6916.07,E2 -6916.07} C_VEL
LIN {X 0,Y 483.061,Z 490.187,A -85,B 0,C 180,E1 -6916.753,E2 -6916.753} C_VEL
LIN {X 0,Y 482.597,Z 501.769,A -85,B 0,C 180,E1 -6917.596,E2 -6917.596} C_VEL
LIN {X 0,Y 482.174,Z 512.223,A -85,B 0,C 180,E1 -6918.545,E2 -6918.545} C_VEL
LIN {X 0,Y 481.818,Z 520.779,A -85,B 0,C 180,E1 -6919.494,E2 -6919.494} C_VEL
LIN {X 0,Y 481.472,Z 528.676,A -85,B 0,C 180,E1 -6920.548,E2 -6920.548} C_VEL
LIN {X 0,Y 481.226,Z 536.395,A -85,B 0,C 180,E1 -6921.813,E2 -6921.813} C_VEL
LIN {X 0,Y 481.005,Z 543.513,A -85,B 0,C 180,E1 -6923.287,E2 -6923.287} C_VEL
LIN {X 0,Y 480.931,Z 548.253,A -85,B 0,C 180,E1 -6924.549,E2 -6924.549} C_VEL
LIN {X 0,Y 480.829,Z 551.873,A -85,B 0,C 180,E1 -6925.808,E2 -6925.808} C_VEL
LIN {X 0,Y 480.888,Z 553.746,A -85,B 0,C 180,E1 -6926.648,E2 -6926.648} C_VEL
LIN {X 0,Y 480.821,Z 556.149,A -85,B 0,C 180,E1 -6928.324,E2 -6928.324} C_VEL
LIN {X 0,Y 480.745,Z 556.978,A -85,B 0,C 180,E1 -6929.999,E2 -6929.999} C_VEL
LIN {X 0,Y 480.821,Z 556.159,A -85,B 0,C 180,E1 -6931.675,E2 -6931.675} C_VEL
LIN {X 0,Y 480.888,Z 553.764,A -85,B 0,C 180,E1 -6933.351,E2 -6933.351} C_VEL
LIN {X 0,Y 480.838,Z 550.817,A -85,B 0,C 180,E1 -6934.61,E2 -6934.61} C_VEL
LIN {X 0,Y 480.925,Z 546.831,A -85,B 0,C 180,E1 -6935.871,E2 -6935.871} C_VEL
LIN {X 0,Y 481.105,Z 540.696,A -85,B 0,C 180,E1 -6937.343,E2 -6937.343} C_VEL
LIN {X 0,Y 481.31,Z 533.992,A -85,B 0,C 180,E1 -6938.607,E2 -6938.607} C_VEL
LIN {X 0,Y 481.592,Z 525.674,A -85,B 0,C 180,E1 -6939.873,E2 -6939.873} C_VEL
LIN {X 0,Y 481.982,Z 517.142,A -85,B 0,C 180,E1 -6940.926,E2 -6940.926} C_VEL
LIN {X 0,Y 482.442,Z 506.6,A -85,B 0,C 180,E1 -6941.98,E2 -6941.98} C_VEL
LIN {X 0,Y 482.867,Z 495.234,A -85,B 0,C 180,E1 -6942.893,E2 -6942.893} C_VEL
LIN {X 0,Y 483.239,Z 484.713,A -85,B 0,C 180,E1 -6943.562,E2 -6943.562} C_VEL
LIN {X 0,Y 483.648,Z 472.896,A -85,B 0,C 180,E1 -6944.14,E2 -6944.14} C_VEL
LIN {X 0,Y 483.976,Z 459.244,A -85,B 0,C 180,E1 -6944.613,E2 -6944.613} C_VEL
LIN {X 0,Y 484.293,Z 447.061,A -85,B 0,C 180,E1 -6944.872,E2 -6944.872} C_VEL
LIN {X 0,Y 484.721,Z 360.274,A -85,B 0,C 180,E1 -6946.168,E2 -6946.168} C_VEL
LIN {X 0,Y 482.254,Z 344.049,A -85,B 0,C 180,E1 -6946.509,E2 -6946.509} C_VEL
LIN {X 0,Y 482.896,Z 325.677,A -85,B 0,C 180,E1 -6949.556,E2 -6949.556} C_VEL
LIN {X 0,Y 483.597,Z 305.889,A -85,B 0,C 180,E1 -6952.876,E2 -6952.876} C_VEL
LIN {X 0,Y 483.67,Z 300.856,A -85,B 0,C 180,E1 -6953.733,E2 -6953.733} C_VEL
LIN {X 0,Y 481.743,Z 290.479,A -85,B 0,C 180,E1 -6955.629,E2 -6955.629} C_VEL
LIN {X 0,Y 481.699,Z 290.485,A -85,B 0,C 180,E1 -6957.831,E2 -6957.831} C_VEL
LIN {X 0,Y 481.643,Z 290.486,A -85,B 0,C 180,E1 -6960.71,E2 -6960.71} C_VEL
LIN {X 0,Y 481.694,Z 290.48,A -85,B 0,C 180,E1 -6963.732,E2 -6963.732} C_VEL
LIN {X 0,Y 481.624,Z 290.489,A -85,B 0,C 180,E1 -6966.746,E2 -6966.746} C_VEL
LIN {X 0,Y 481.672,Z 290.484,A -85,B 0,C 180,E1 -6969.939,E2 -6969.939} C_VEL
LIN {X 0,Y 481.634,Z 290.485,A -85,B 0,C 180,E1 -6973.299,E2 -6973.299} C_VEL
LIN {X 0,Y 481.654,Z 290.483,A -85,B 0,C 180,E1 -6975.64,E2 -6975.64} C_VEL
LIN {X 0,Y 481.657,Z 290.486,A -85,B 0,C 180,E1 -6978.958,E2 -6978.958} C_VEL
LIN {X 0,Y 481.65,Z 290.484,A -85,B 0,C 180,E1 -6981.991,E2 -6981.991} C_VEL
LIN {X 0,Y 481.684,Z 290.48,A -85,B 0,C 180,E1 -6985.317,E2 -6985.317} C_VEL
LIN {X 0,Y 481.648,Z 290.485,A -85,B 0,C 180,E1 -6988.312,E2 -6988.312} C_VEL
LIN {X 0,Y 481.697,Z 290.482,A -85,B 0,C 180,E1 -6991.218,E2 -6991.218} C_VEL
LIN {X 0,Y 481.698,Z 290.477,A -85,B 0,C 180,E1 -6994.043,E2 -6994.043} C_VEL
LIN {X 0,Y 481.665,Z 290.486,A -85,B 0,C 180,E1 -6996.811,E2 -6996.811} C_VEL
LIN {X 0,Y 481.686,Z 290.482,A -85,B 0,C 180,E1 -6999.502,E2 -6999.502} C_VEL
LIN {X 0,Y 481.697,Z 290.477,A -85,B 0,C 180,E1 -7002.158,E2 -7002.158} C_VEL
LIN {X 0,Y 481.734,Z 290.475,A -85,B 0,C 180,E1 -7004.776,E2 -7004.776} C_VEL
LIN {X 0,Y 481.743,Z 290.472,A -85,B 0,C 180,E1 -7008.215,E2 -7008.215} C_VEL
LIN {X 0,Y 481.754,Z 290.477,A -85,B 0,C 180,E1 -7011.612,E2 -7011.612} C_VEL
LIN {X 0,Y 481.806,Z 290.465,A -85,B 0,C 180,E1 -7014.139,E2 -7014.139} C_VEL
LIN {X 0,Y 481.917,Z 290.457,A -85,B 0,C 180,E1 -7017.493,E2 -7017.493} C_VEL
LIN {X 0,Y 481.895,Z 290.453,A -85,B 0,C 180,E1 -7020.836,E2 -7020.836} C_VEL
LIN {X 0,Y 481.918,Z 290.45,A -85,B 0,C 180,E1 -7022.508,E2 -7022.508} C_VEL
LIN {X 0,Y 481.789,Z 290.475,A -85,B 0,C 180,E1 -7025.861,E2 -7025.861} C_VEL
LIN {X 0,Y 481.753,Z 290.473,A -85,B 0,C 180,E1 -7028.389,E2 -7028.389} C_VEL
LIN {X 0,Y 481.741,Z 290.478,A -85,B 0,C 180,E1 -7031.785,E2 -7031.785} C_VEL
LIN {X 0,Y 481.732,Z 290.473,A -85,B 0,C 180,E1 -7035.225,E2 -7035.225} C_VEL
LIN {X 0,Y 481.703,Z 290.478,A -85,B 0,C 180,E1 -7038.722,E2 -7038.722} C_VEL
LIN {X 0,Y 481.636,Z 290.485,A -85,B 0,C 180,E1 -7041.395,E2 -7041.395} C_VEL
LIN {X 0,Y 481.648,Z 290.489,A -85,B 0,C 180,E1 -7044.115,E2 -7044.115} C_VEL
LIN {X 0,Y 481.704,Z 290.477,A -85,B 0,C 180,E1 -7047.132,E2 -7047.132} C_VEL
LIN {X 0,Y 481.67,Z 290.481,A -85,B 0,C 180,E1 -7049.742,E2 -7049.742} C_VEL
LIN {X 0,Y 481.664,Z 290.489,A -85,B 0,C 180,E1 -7052.675,E2 -7052.675} C_VEL
LIN {X 0,Y 481.629,Z 290.486,A -85,B 0,C 180,E1 -7055.71,E2 -7055.71} C_VEL
LIN {X 0,Y 481.659,Z 290.489,A -85,B 0,C 180,E1 -7058.86,E2 -7058.86} C_VEL
LIN {X 0,Y 481.633,Z 290.486,A -85,B 0,C 180,E1 -7062.163,E2 -7062.163} C_VEL
LIN {X 0,Y 481.648,Z 290.484,A -85,B 0,C 180,E1 -7065.543,E2 -7065.543} C_VEL
LIN {X 0,Y 481.626,Z 290.495,A -85,B 0,C 180,E1 -7068.957,E2 -7068.957} C_VEL
LIN {X 0,Y 481.644,Z 290.484,A -85,B 0,C 180,E1 -7071.995,E2 -7071.995} C_VEL
LIN {X 0,Y 481.68,Z 290.486,A -85,B 0,C 180,E1 -7075.318,E2 -7075.318} C_VEL
LIN {X 0,Y 481.637,Z 290.485,A -85,B 0,C 180,E1 -7078.312,E2 -7078.312} C_VEL
LIN {X 0,Y 481.656,Z 290.49,A -85,B 0,C 180,E1 -7081.217,E2 -7081.217} C_VEL
LIN {X 0,Y 481.628,Z 290.486,A -85,B 0,C 180,E1 -7084.331,E2 -7084.331} C_VEL
LIN {X 0,Y 481.653,Z 290.484,A -85,B 0,C 180,E1 -7086.819,E2 -7086.819} C_VEL
LIN {X 0,Y 481.635,Z 290.487,A -85,B 0,C 180,E1 -7087.966,E2 -7087.966} C_VEL
LIN {X 0,Y 480.968,Z 290.569,A -85,B 0,C 180,E1 -7088.664,E2 -7088.664} C_VEL
LIN {X 0,Y 478.144,Z 290.925,A -85,B 0,C 180,E1 -7089.798,E2 -7089.798} C_VEL
LIN {X 0,Y 475.758,Z 291.223,A -85,B 0,C 180,E1 -7090.712,E2 -7090.712} C_VEL
LIN {X 0,Y 474.729,Z 291.352,A -85,B 0,C 180,E1 -7091.418,E2 -7091.418} C_VEL
LIN {X 0,Y 474.643,Z 291.361,A -85,B 0,C 180,E1 -7091.657,E2 -7091.657} C_VEL
LIN {X 0,Y 474.698,Z 291.349,A -85,B 0,C 180,E1 -7094.545,E2 -7094.545} C_VEL
LIN {X 0,Y 474.677,Z 291.356,A -85,B 0,C 180,E1 -7098.038,E2 -7098.038} C_VEL
LIN {X 0,Y 474.661,Z 291.361,A -85,B 0,C 180,E1 -7101.486,E2 -7101.486} C_VEL
LIN {X 0,Y 474.725,Z 291.449,A -85,B 0,C 180,E1 -7103.466,E2 -7103.466} C_VEL
LIN {X 0,Y 475.529,Z 297.407,A -85,B 0,C 180,E1 -7104.701,E2 -7104.701} C_VEL
LIN {X 0,Y 475.336,Z 309.157,A -85,B 0,C 180,E1 -7107.034,E2 -7107.034} C_VEL
LIN {X 0,Y 475.326,Z 310.698,A -85,B 0,C 180,E1 -7107.339,E2 -7107.339} C_VEL
LIN {X 0,Y 478.122,Z 325.116,A -85,B 0,C 180,E1 -7107.658,E2 -7107.658} C_VEL
LIN {X 0,Y 477.412,Z 417.865,A -85,B 0,C 180,E1 -7109.078,E2 -7109.078} C_VEL
LIN {X 0,Y 477.131,Z 430.968,A -85,B 0,C 180,E1 -7109.447,E2 -7109.447} C_VEL
LIN {X 0,Y 476.821,Z 442.985,A -85,B 0,C 180,E1 -7109.948,E2 -7109.948} C_VEL
LIN {X 0,Y 476.424,Z 455.162,A -85,B 0,C 180,E1 -7110.635,E2 -7110.635} C_VEL
LIN {X 0,Y 475.936,Z 466.669,A -85,B 0,C 180,E1 -7111.481,E2 -7111.481} C_VEL
LIN {X 0,Y 475.451,Z 477.039,A -85,B 0,C 180,E1 -7112.436,E2 -7112.436} C_VEL
LIN {X 0,Y 475.027,Z 485.535,A -85,B 0,C 180,E1 -7113.393,E2 -7113.393} C_VEL
LIN {X 0,Y 474.696,Z 493.367,A -85,B 0,C 180,E1 -7114.459,E2 -7114.459} C_VEL
LIN {X 0,Y 474.357,Z 501.043,A -85,B 0,C 180,E1 -7115.74,E2 -7115.74} C_VEL
LIN {X 0,Y 474.224,Z 506.288,A -85,B 0,C 180,E1 -7116.81,E2 -7116.81} C_VEL
LIN {X 0,Y 474.008,Z 511.397,A -85,B 0,C 180,E1 -7118.098,E2 -7118.098} C_VEL
LIN {X 0,Y 473.862,Z 515.368,A -85,B 0,C 180,E1 -7119.39,E2 -7119.39} C_VEL
LIN {X 0,Y 473.805,Z 517.41,A -85,B 0,C 180,E1 -7120.254,E2 -7120.254} C_VEL
LIN {X 0,Y 473.737,Z 519.912,A -85,B 0,C 180,E1 -7121.726,E2 -7121.726} C_VEL
LIN {X 0,Y 473.667,Z 521.015,A -85,B 0,C 180,E1 -7122.86,E2 -7122.86} C_VEL
LIN {X 0,Y 473.635,Z 521.373,A -85,B 0,C 180,E1 -7123.734,E2 -7123.734} C_VEL
LIN {X 0,Y 473.665,Z 520.985,A -85,B 0,C 180,E1 -7125.325,E2 -7125.325} C_VEL
LIN {X 0,Y 473.634,Z 519.949,A -85,B 0,C 180,E1 -7126.376,E2 -7126.376} C_VEL
LIN {X 0,Y 473.705,Z 518.612,A -85,B 0,C 180,E1 -7127.261,E2 -7127.261} C_VEL
LIN {X 0,Y 473.84,Z 516.386,A -85,B 0,C 180,E1 -7128.332,E2 -7128.332} C_VEL
LIN {X 0,Y 473.998,Z 511.726,A -85,B 0,C 180,E1 -7129.94,E2 -7129.94} C_VEL
LIN {X 0,Y 474.213,Z 506.379,A -85,B 0,C 180,E1 -7131.309,E2 -7131.309} C_VEL
LIN {X 0,Y 474.473,Z 499.663,A -85,B 0,C 180,E1 -7132.651,E2 -7132.651} C_VEL
LIN {X 0,Y 474.903,Z 491.085,A -85,B 0,C 180,E1 -7134.015,E2 -7134.015} C_VEL
LIN {X 0,Y 475.337,Z 482.169,A -85,B 0,C 180,E1 -7135.156,E2 -7135.156} C_VEL
LIN {X 0,Y 475.751,Z 471.99,A -85,B 0,C 180,E1 -7136.206,E2 -7136.206} C_VEL
LIN {X 0,Y 476.314,Z 461.158,A -85,B 0,C 180,E1 -7137.101,E2 -7137.101} C_VEL
LIN {X 0,Y 476.729,Z 450.489,A -85,B 0,C 180,E1 -7137.806,E2 -7137.806} C_VEL
LIN {X 0,Y 477.058,Z 438.273,A -85,B 0,C 180,E1 -7138.426,E2 -7138.426} C_VEL
LIN {X 0,Y 477.32,Z 425.393,A -85,B 0,C 180,E1 -7138.89,E2 -7138.89} C_VEL
LIN {X 0,Y 477.534,Z 412.087,A -85,B 0,C 180,E1 -7139.187,E2 -7139.187} C_VEL
LIN {X 0,Y 478.214,Z 324.518,A -85,B 0,C 180,E1 -7140.52,E2 -7140.52} C_VEL
LIN {X 0,Y 475.413,Z 310.516,A -85,B 0,C 180,E1 -7140.874,E2 -7140.874} C_VEL
LIN {X 0,Y 475.645,Z 297.409,A -85,B 0,C 180,E1 -7143.394,E2 -7143.394} C_VEL
LIN {X 0,Y 474.681,Z 291.36,A -85,B 0,C 180,E1 -7144.623,E2 -7144.623} C_VEL
LIN {X 0,Y 474.612,Z 291.367,A -85,B 0,C 180,E1 -7148.296,E2 -7148.296} C_VEL
LIN {X 0,Y 474.63,Z 291.362,A -85,B 0,C 180,E1 -7150.959,E2 -7150.959} C_VEL
LIN {X 0,Y 474.608,Z 291.367,A -85,B 0,C 180,E1 -7154.105,E2 -7154.105} C_VEL
LIN {X 0,Y 474.616,Z 291.365,A -85,B 0,C 180,E1 -7157.066,E2 -7157.066} C_VEL
LIN {X 0,Y 474.646,Z 291.359,A -85,B 0,C 180,E1 -7160.454,E2 -7160.454} C_VEL
LIN {X 0,Y 474.59,Z 291.364,A -85,B 0,C 180,E1 -7163.676,E2 -7163.676} C_VEL
LIN {X 0,Y 474.644,Z 291.363,A -85,B 0,C 180,E1 -7166.78,E2 -7166.78} C_VEL
LIN {X 0,Y 474.606,Z 291.359,A -85,B 0,C 180,E1 -7169.77,E2 -7169.77} C_VEL
LIN {X 0,Y 474.698,Z 291.353,A -85,B 0,C 180,E1 -7172.68,E2 -7172.68} C_VEL
LIN {X 0,Y 474.657,Z 291.358,A -85,B 0,C 180,E1 -7175.507,E2 -7175.507} C_VEL
LIN {X 0,Y 474.671,Z 291.36,A -85,B 0,C 180,E1 -7179.185,E2 -7179.185} C_VEL
LIN {X 0,Y 474.656,Z 291.356,A -85,B 0,C 180,E1 -7181.884,E2 -7181.884} C_VEL
LIN {X 0,Y 474.7,Z 291.348,A -85,B 0,C 180,E1 -7184.544,E2 -7184.544} C_VEL
LIN {X 0,Y 474.704,Z 291.352,A -85,B 0,C 180,E1 -7188.037,E2 -7188.037} C_VEL
LIN {X 0,Y 474.727,Z 291.346,A -85,B 0,C 180,E1 -7191.486,E2 -7191.486} C_VEL
LIN {X 0,Y 474.769,Z 291.343,A -85,B 0,C 180,E1 -7194.052,E2 -7194.052} C_VEL
LIN {X 0,Y 474.893,Z 291.326,A -85,B 0,C 180,E1 -7197.455,E2 -7197.455} C_VEL
LIN {X 0,Y 474.911,Z 291.325,A -85,B 0,C 180,E1 -7200,E2 -7200} C_VEL
LIN {X 0,Y 474.893,Z 291.327,A -85,B 0,C 180,E1 -7202.545,E2 -7202.545} C_VEL
LIN {X 0,Y 474.769,Z 291.342,A -85,B 0,C 180,E1 -7205.948,E2 -7205.948} C_VEL
LIN {X 0,Y 474.726,Z 291.35,A -85,B 0,C 180,E1 -7208.514,E2 -7208.514} C_VEL
LIN {X 0,Y 474.704,Z 291.346,A -85,B 0,C 180,E1 -7211.962,E2 -7211.962} C_VEL
LIN {X 0,Y 474.7,Z 291.346,A -85,B 0,C 180,E1 -7215.456,E2 -7215.456} C_VEL
LIN {X 0,Y 474.665,Z 291.356,A -85,B 0,C 180,E1 -7219.01,E2 -7219.01} C_VEL
LIN {X 0,Y 474.588,Z 291.36,A -85,B 0,C 180,E1 -7221.729,E2 -7221.729} C_VEL
LIN {X 0,Y 474.655,Z 291.361,A -85,B 0,C 180,E1 -7224.493,E2 -7224.493} C_VEL
LIN {X 0,Y 474.681,Z 291.354,A -85,B 0,C 180,E1 -7227.334,E2 -7227.334} C_VEL
LIN {X 0,Y 474.605,Z 291.358,A -85,B 0,C 180,E1 -7230.23,E2 -7230.23} C_VEL
LIN {X 0,Y 474.625,Z 291.361,A -85,B 0,C 180,E1 -7233.222,E2 -7233.222} C_VEL
LIN {X 0,Y 474.589,Z 291.364,A -85,B 0,C 180,E1 -7236.324,E2 -7236.324} C_VEL
LIN {X 0,Y 474.619,Z 291.362,A -85,B 0,C 180,E1 -7239.646,E2 -7239.646} C_VEL
LIN {X 0,Y 474.616,Z 291.364,A -85,B 0,C 180,E1 -7242.934,E2 -7242.934} C_VEL
LIN {X 0,Y 474.607,Z 291.364,A -85,B 0,C 180,E1 -7245.895,E2 -7245.895} C_VEL
LIN {X 0,Y 474.629,Z 291.362,A -85,B 0,C 180,E1 -7249.041,E2 -7249.041} C_VEL
LIN {X 0,Y 474.612,Z 291.366,A -85,B 0,C 180,E1 -7251.704,E2 -7251.704} C_VEL
LIN {X 0,Y 474.626,Z 291.36,A -85,B 0,C 180,E1 -7254.726,E2 -7254.726} C_VEL
LIN {X 0,Y 474.638,Z 291.365,A -85,B 0,C 180,E1 -7257.788,E2 -7257.788} C_VEL
LIN {X 0,Y 474.626,Z 291.361,A -85,B 0,C 180,E1 -7260.885,E2 -7260.885} C_VEL
LIN {X 0,Y 474.674,Z 291.359,A -85,B 0,C 180,E1 -7263.629,E2 -7263.629} C_VEL
LIN {X 0,Y 474.715,Z 291.544,A -85,B 0,C 180,E1 -7264.104,E2 -7264.104} C_VEL
LIN {X 0,Y 476.815,Z 302.789,A -85,B 0,C 180,E1 -7266.216,E2 -7266.216} C_VEL
LIN {X 0,Y 476.383,Z 315.095,A -85,B 0,C 180,E1 -7268.346,E2 -7268.346} C_VEL
LIN {X 0,Y 475.685,Z 333.493,A -85,B 0,C 180,E1 -7271.479,E2 -7271.479} C_VEL
LIN {X 0,Y 475.279,Z 343.647,A -85,B 0,C 180,E1 -7273.189,E2 -7273.189} C_VEL
LIN {X 0,Y 478.064,Z 361.365,A -85,B 0,C 180,E1 -7273.571,E2 -7273.571} C_VEL
LIN {X 0,Y 477.423,Z 451.827,A -85,B 0,C 180,E1 -7274.962,E2 -7274.962} C_VEL
LIN {X 0,Y 477.094,Z 465.174,A -85,B 0,C 180,E1 -7275.333,E2 -7275.333} C_VEL
LIN {X 0,Y 476.646,Z 477.942,A -85,B 0,C 180,E1 -7275.864,E2 -7275.864} C_VEL
LIN {X 0,Y 476.126,Z 490.1,A -85,B 0,C 180,E1 -7276.557,E2 -7276.557} C_VEL
LIN {X 0,Y 475.683,Z 500.89,A -85,B 0,C 180,E1 -7277.349,E2 -7277.349} C_VEL
LIN {X 0,Y 475.265,Z 510.992,A -85,B 0,C 180,E1 -7278.268,E2 -7278.268} C_VEL
LIN {X 0,Y 474.814,Z 520.589,A -85,B 0,C 180,E1 -7279.337,E2 -7279.337} C_VEL
LIN {X 0,Y 474.37,Z 529.837,A -85,B 0,C 180,E1 -7280.62,E2 -7280.62} C_VEL
LIN {X 0,Y 474.114,Z 537.28,A -85,B 0,C 180,E1 -7281.904,E2 -7281.904} C_VEL
LIN {X 0,Y 473.922,Z 543.262,A -85,B 0,C 180,E1 -7283.186,E2 -7283.186} C_VEL
LIN {X 0,Y 473.845,Z 547.999,A -85,B 0,C 180,E1 -7284.467,E2 -7284.467} C_VEL
LIN {X 0,Y 473.735,Z 551.617,A -85,B 0,C 180,E1 -7285.746,E2 -7285.746} C_VEL
LIN {X 0,Y 473.795,Z 553.487,A -85,B 0,C 180,E1 -7286.598,E2 -7286.598} C_VEL
LIN {X 0,Y 473.724,Z 555.887,A -85,B 0,C 180,E1 -7288.299,E2 -7288.299} C_VEL
LIN {X 0,Y 473.688,Z 556.498,A -85,B 0,C 180,E1 -7289.149,E2 -7289.149} C_VEL
LIN {X 0,Y 473.672,Z 556.714,A -85,B 0,C 180,E1 -7289.999,E2 -7289.999} C_VEL
LIN {X 0,Y 473.724,Z 555.89,A -85,B 0,C 180,E1 -7291.7,E2 -7291.7} C_VEL
LIN {X 0,Y 473.741,Z 554.893,A -85,B 0,C 180,E1 -7292.55,E2 -7292.55} C_VEL
LIN {X 0,Y 473.795,Z 553.491,A -85,B 0,C 180,E1 -7293.401,E2 -7293.401} C_VEL
LIN {X 0,Y 473.761,Z 550.541,A -85,B 0,C 180,E1 -7294.679,E2 -7294.679} C_VEL
LIN {X 0,Y 473.832,Z 546.55,A -85,B 0,C 180,E1 -7295.959,E2 -7295.959} C_VEL
LIN {X 0,Y 474.014,Z 540.407,A -85,B 0,C 180,E1 -7297.453,E2 -7297.453} C_VEL
LIN {X 0,Y 474.259,Z 533.697,A -85,B 0,C 180,E1 -7298.736,E2 -7298.736} C_VEL
LIN {X 0,Y 474.556,Z 525.36,A -85,B 0,C 180,E1 -7300.02,E2 -7300.02} C_VEL
LIN {X 0,Y 474.966,Z 516.8,A -85,B 0,C 180,E1 -7301.09,E2 -7301.09} C_VEL
LIN {X 0,Y 475.443,Z 506.426,A -85,B 0,C 180,E1 -7302.141,E2 -7302.141} C_VEL
LIN {X 0,Y 475.911,Z 494.452,A -85,B 0,C 180,E1 -7303.111,E2 -7303.111} C_VEL
LIN {X 0,Y 476.376,Z 482.244,A -85,B 0,C 180,E1 -7303.87,E2 -7303.87} C_VEL
LIN {X 0,Y 476.863,Z 469.688,A -85,B 0,C 180,E1 -7304.454,E2 -7304.454} C_VEL
LIN {X 0,Y 477.162,Z 457.577,A -85,B 0,C 180,E1 -7304.854,E2 -7304.854} C_VEL
LIN {X 0,Y 477.419,Z 444.139,A -85,B 0,C 180,E1 -7305.119,E2 -7305.119} C_VEL
LIN {X 0,Y 477.925,Z 361.354,A -85,B 0,C 180,E1 -7306.37,E2 -7306.37} C_VEL
LIN {X 0,Y 475.235,Z 343.871,A -85,B 0,C 180,E1 -7306.731,E2 -7306.731} C_VEL
LIN {X 0,Y 475.896,Z 326.752,A -85,B 0,C 180,E1 -7309.608,E2 -7309.608} C_VEL
LIN {X 0,Y 476.655,Z 306.822,A -85,B 0,C 180,E1 -7312.999,E2 -7312.999} C_VEL
LIN {X 0,Y 476.628,Z 301.601,A -85,B 0,C 180,E1 -7313.906,E2 -7313.906} C_VEL
LIN {X 0,Y 474.701,Z 291.357,A -85,B 0,C 180,E1 -7315.83,E2 -7315.83} C_VEL
LIN {X 0,Y 474.644,Z 291.365,A -85,B 0,C 180,E1 -7318.281,E2 -7318.281} C_VEL
LIN {X 0,Y 474.596,Z 291.362,A -85,B 0,C 180,E1 -7321.217,E2 -7321.217} C_VEL
LIN {X 0,Y 474.631,Z 291.366,A -85,B 0,C 180,E1 -7324.24,E2 -7324.24} C_VEL
LIN {X 0,Y 474.587,Z 291.363,A -85,B 0,C 180,E1 -7327.383,E2 -7327.383} C_VEL
LIN {X 0,Y 474.612,Z 291.364,A -85,B 0,C 180,E1 -7330.657,E2 -7330.657} C_VEL
LIN {X 0,Y 474.597,Z 291.362,A -85,B 0,C 180,E1 -7333.48,E2 -7333.48} C_VEL
LIN {X 0,Y 474.616,Z 291.369,A -85,B 0,C 180,E1 -7336.515,E2 -7336.515} C_VEL
LIN {X 0,Y 474.613,Z 291.36,A -85,B 0,C 180,E1 -7339.342,E2 -7339.342} C_VEL
LIN {X 0,Y 474.605,Z 291.361,A -85,B 0,C 180,E1 -7341.703,E2 -7341.703} C_VEL
LIN {X 0,Y 474.622,Z 291.368,A -85,B 0,C 180,E1 -7344.725,E2 -7344.725} C_VEL
LIN {X 0,Y 474.63,Z 291.357,A -85,B 0,C 180,E1 -7347.787,E2 -7347.787} C_VEL
LIN {X 0,Y 474.624,Z 291.367,A -85,B 0,C 180,E1 -7350.882,E2 -7350.882} C_VEL
LIN {X 0,Y 474.658,Z 291.355,A -85,B 0,C 180,E1 -7353.628,E2 -7353.628} C_VEL
LIN {X 0,Y 474.627,Z 291.361,A -85,B 0,C 180,E1 -7356.641,E2 -7356.641} C_VEL
LIN {X 0,Y 474.645,Z 291.356,A -85,B 0,C 180,E1 -7360.089,E2 -7360.089} C_VEL
LIN {X 0,Y 474.641,Z 291.359,A -85,B 0,C 180,E1 -7362.774,E2 -7362.774} C_VEL
LIN {X 0,Y 474.643,Z 291.363,A -85,B 0,C 180,E1 -7365.421,E2 -7365.421} C_VEL
LIN {X 0,Y 474.696,Z 291.35,A -85,B 0,C 180,E1 -7368.037,E2 -7368.037} C_VEL
LIN {X 0,Y 474.719,Z 291.355,A -85,B 0,C 180,E1 -7371.486,E2 -7371.486} C_VEL
LIN {X 0,Y 474.769,Z 291.342,A -85,B 0,C 180,E1 -7374.052,E2 -7374.052} C_VEL
LIN {X 0,Y 474.884,Z 291.333,A -85,B 0,C 180,E1 -7377.455,E2 -7377.455} C_VEL
